F_ADD_STRINGX4_TO_BUFFER( S1:= CONCAT(sHead, '_EVP0_mA' ), S2:='$t', S3:= REAL_TO_STRING( stPropulsionCfg.aEVP_mA[0]  ), S4:='$n', wSize := wSize, pBuffer := pBuffer, wPos := wBufPos );
F_ADD_STRINGX4_TO_BUFFER( S1:= CONCAT(sHead, '_EVP1_mA' ), S2:='$t', S3:= REAL_TO_STRING( stPropulsionCfg.aEVP_mA[1]  ), S4:='$n', wSize := wSize, pBuffer := pBuffer, wPos := wBufPos );
F_ADD_STRINGX4_TO_BUFFER( S1:= CONCAT(sHead, '_EVP2_mA' ), S2:='$t', S3:= REAL_TO_STRING( stPropulsionCfg.aEVP_mA[2]  ), S4:='$n', wSize := wSize, pBuffer := pBuffer, wPos := wBufPos );
F_ADD_STRINGX4_TO_BUFFER( S1:= CONCAT(sHead, '_EVP3_mA' ), S2:='$t', S3:= REAL_TO_STRING( stPropulsionCfg.aEVP_mA[3]  ), S4:='$n', wSize := wSize, pBuffer := pBuffer, wPos := wBufPos );
F_ADD_STRINGX4_TO_BUFFER( S1:= CONCAT(sHead, '_EVP4_mA' ), S2:='$t', S3:= REAL_TO_STRING( stPropulsionCfg.aEVP_mA[4]  ), S4:='$n', wSize := wSize, pBuffer := pBuffer, wPos := wBufPos );
F_ADD_STRINGX4_TO_BUFFER( S1:= CONCAT(sHead, '_EVP5_mA' ), S2:='$t', S3:= REAL_TO_STRING( 0.0                         ), S4:='$n', wSize := wSize, pBuffer := pBuffer, wPos := wBufPos );
F_ADD_STRINGX4_TO_BUFFER( S1:= CONCAT(sHead, '_EVP6_mA' ), S2:='$t', S3:= REAL_TO_STRING( stPropulsionCfg.aEVP_mA[6]  ), S4:='$n', wSize := wSize, pBuffer := pBuffer, wPos := wBufPos );
F_ADD_STRINGX4_TO_BUFFER( S1:= CONCAT(sHead, '_EVP7_mA' ), S2:='$t', S3:= REAL_TO_STRING( stPropulsionCfg.aEVP_mA[7]  ), S4:='$n', wSize := wSize, pBuffer := pBuffer, wPos := wBufPos );
F_ADD_STRINGX4_TO_BUFFER( S1:= CONCAT(sHead, '_EVP8_mA' ), S2:='$t', S3:= REAL_TO_STRING( stPropulsionCfg.aEVP_mA[8]  ), S4:='$n', wSize := wSize, pBuffer := pBuffer, wPos := wBufPos );
F_ADD_STRINGX4_TO_BUFFER( S1:= CONCAT(sHead, '_EVP9_mA' ), S2:='$t', S3:= REAL_TO_STRING( stPropulsionCfg.aEVP_mA[9]  ), S4:='$n', wSize := wSize, pBuffer := pBuffer, wPos := wBufPos );
F_ADD_STRINGX4_TO_BUFFER( S1:= CONCAT(sHead, '_EVP10_mA'), S2:='$t', S3:= REAL_TO_STRING( stPropulsionCfg.aEVP_mA[10] ), S4:='$n', wSize := wSize, pBuffer := pBuffer, wPos := wBufPos );
END_FUNCTION

(* POU FUN/PARAMETERS/F_WRITE_SE_CYLINDER_POS_CFG, ST *)
FUNCTION F_WRITE_SE_CYLINDER_POS_CFG : BOOL
VAR_INPUT
	sHead : STRING;
	wSize   :DWORD;
	pBuffer :POINTER TO BYTE;
END_VAR
VAR_IN_OUT
	wPos     : DWORD;
	stConfig : ST_SE_CYLINDER_POS_CFG;
END_VAR
VAR
END_VAR
F_ADD_STRINGX3_TO_BUFFER( S1:= '$n#', S2:= sHead, S3:=' - Parameters:$n', wSize := wSize, pBuffer := pBuffer, wPos := wPos );

F_ADD_STRINGX4_TO_BUFFER( S1:= CONCAT(sHead, '_Ease'    ), S2:='$t', S3:= REAL_TO_STRING( stConfig.Ease    ), S4:='$n', wSize := wSize, pBuffer := pBuffer, wPos := wPos );

F_ADD_STRINGX4_TO_BUFFER( S1:= CONCAT(sHead, '_TgtLS_In'  ), S2:='$t', S3:= REAL_TO_STRING( stConfig.TgtLS_In  ), S4:='$n', wSize := wSize, pBuffer := pBuffer, wPos := wPos );
F_ADD_STRINGX4_TO_BUFFER( S1:= CONCAT(sHead, '_TgtLS_Out' ), S2:='$t', S3:= REAL_TO_STRING( stConfig.TgtLS_Out ), S4:='$n', wSize := wSize, pBuffer := pBuffer, wPos := wPos );
F_ADD_STRINGX4_TO_BUFFER( S1:= CONCAT(sHead, '_TgtLS_Slow' ), S2:='$t', S3:= REAL_TO_STRING( stConfig.TgtLS_Slow ), S4:='$n', wSize := wSize, pBuffer := pBuffer, wPos := wPos );

F_ADD_STRINGX4_TO_BUFFER( S1:= CONCAT(sHead, '_TimeMax'  ), S2:='$t', S3:= REAL_TO_STRING( stConfig.TimeMax  ), S4:='$n', wSize := wSize, pBuffer := pBuffer, wPos := wPos );
F_ADD_STRINGX4_TO_BUFFER( S1:= CONCAT(sHead, '_TimeEase' ), S2:='$t', S3:= REAL_TO_STRING( stConfig.TimeEase ), S4:='$n', wSize := wSize, pBuffer := pBuffer, wPos := wPos );

F_ADD_STRINGX4_TO_BUFFER( S1:= CONCAT(sHead, '_LS_Limit_In'  ), S2:='$t', S3:= BOOL_TO_STRING( stConfig.LS_Limit_In  ), S4:='$n', wSize := wSize, pBuffer := pBuffer, wPos := wPos );
F_ADD_STRINGX4_TO_BUFFER( S1:= CONCAT(sHead, '_LS_Limit_Out' ), S2:='$t', S3:= BOOL_TO_STRING( stConfig.LS_Limit_Out ), S4:='$n', wSize := wSize, pBuffer := pBuffer, wPos := wPos );

F_ADD_STRINGX4_TO_BUFFER( S1:= CONCAT(sHead, '_HP'  ), S2:='$t', S3:= BYTE_TO_STRING( stConfig.HP ), S4:='$n', wSize := wSize, pBuffer := pBuffer, wPos := wPos );
END_FUNCTION

(* POU FUN/PARAMETERS/F_WRITE_SE_CYLINDER_CFG, ST *)
FUNCTION F_WRITE_SE_CYLINDER_CFG : BOOL
VAR_INPUT
	sHead : STRING;
	wSize   :DWORD;
	pBuffer :POINTER TO BYTE;
END_VAR
VAR_IN_OUT
	wPos     : DWORD;
	stConfig : ST_SE_CYLINDER_CFG;
END_VAR
VAR
END_VAR
F_ADD_STRINGX3_TO_BUFFER( S1:= '$n#', S2:= sHead, S3:=' - Parameters:$n', wSize := wSize, pBuffer := pBuffer, wPos := wPos );

F_ADD_STRINGX4_TO_BUFFER( S1:= CONCAT(sHead, '_Ease'     ), S2:='$t', S3:= REAL_TO_STRING( stConfig.Ease     ), S4:='$n', wSize := wSize, pBuffer := pBuffer, wPos := wPos );
F_ADD_STRINGX4_TO_BUFFER( S1:= CONCAT(sHead, '_TimeMax'  ), S2:='$t', S3:= REAL_TO_STRING( stConfig.TimeMax  ), S4:='$n', wSize := wSize, pBuffer := pBuffer, wPos := wPos );
F_ADD_STRINGX4_TO_BUFFER( S1:= CONCAT(sHead, '_TimeEase' ), S2:='$t', S3:= REAL_TO_STRING( stConfig.TimeEase ), S4:='$n', wSize := wSize, pBuffer := pBuffer, wPos := wPos );
F_ADD_STRINGX4_TO_BUFFER( S1:= CONCAT(sHead, '_HP'       ), S2:='$t', S3:= BYTE_TO_STRING( stConfig.HP       ), S4:='$n', wSize := wSize, pBuffer := pBuffer, wPos := wPos );
END_FUNCTION

(* POU FUN/PARAMETERS/F_WRITE_LIFT_PROP_CFG, ST *)
FUNCTION F_WRITE_LIFT_PROP_CFG : BOOL
VAR_INPUT
	sHead : STRING;
	wSize   :DWORD;
	pBuffer :POINTER TO BYTE;
END_VAR
VAR_IN_OUT
	wPos     : DWORD;
	stConfig : ST_LIFT_PROP_CFG;
END_VAR
VAR
END_VAR
F_ADD_STRINGX3_TO_BUFFER( S1:= '$n#', S2:= sHead, S3:=' - Parameters:$n', wSize := wSize, pBuffer := pBuffer, wPos := wPos );

F_ADD_STRINGX4_TO_BUFFER( S1:= CONCAT(sHead, '_TgtP_Up'  ), S2:='$t', S3:= REAL_TO_STRING( stConfig.TgtP_Up  ), S4:='$n', wSize := wSize, pBuffer := pBuffer, wPos := wPos );
F_ADD_STRINGX4_TO_BUFFER( S1:= CONCAT(sHead, '_TgtP_Dw'  ), S2:='$t', S3:= REAL_TO_STRING( stConfig.TgtP_Dw  ), S4:='$n', wSize := wSize, pBuffer := pBuffer, wPos := wPos );
F_ADD_STRINGX4_TO_BUFFER( S1:= CONCAT(sHead, '_TgtLS_Up' ), S2:='$t', S3:= REAL_TO_STRING( stConfig.TgtLS_Up ), S4:='$n', wSize := wSize, pBuffer := pBuffer, wPos := wPos );
F_ADD_STRINGX4_TO_BUFFER( S1:= CONCAT(sHead, '_TgtLS_Dw' ), S2:='$t', S3:= REAL_TO_STRING( stConfig.TgtLS_Dw ), S4:='$n', wSize := wSize, pBuffer := pBuffer, wPos := wPos );

F_ADD_STRINGX4_TO_BUFFER( S1:= CONCAT(sHead, '_P_DB'     ), S2:='$t', S3:= REAL_TO_STRING( stConfig.P_DB     ), S4:='$n', wSize := wSize, pBuffer := pBuffer, wPos := wPos );
F_ADD_STRINGX4_TO_BUFFER( S1:= CONCAT(sHead, '_LS_DB'    ), S2:='$t', S3:= REAL_TO_STRING( stConfig.LS_DB    ), S4:='$n', wSize := wSize, pBuffer := pBuffer, wPos := wPos );

F_ADD_STRINGX4_TO_BUFFER( S1:= CONCAT(sHead, '_TimeMax'  ), S2:='$t', S3:= REAL_TO_STRING( stConfig.TimeMax  ), S4:='$n', wSize := wSize, pBuffer := pBuffer, wPos := wPos );
F_ADD_STRINGX4_TO_BUFFER( S1:= CONCAT(sHead, '_Delay_Up' ), S2:='$t', S3:= REAL_TO_STRING( stConfig.Delay_Up ), S4:='$n', wSize := wSize, pBuffer := pBuffer, wPos := wPos );
F_ADD_STRINGX4_TO_BUFFER( S1:= CONCAT(sHead, '_Delay_Dw' ), S2:='$t', S3:= REAL_TO_STRING( stConfig.Delay_Dw ), S4:='$n', wSize := wSize, pBuffer := pBuffer, wPos := wPos );

F_ADD_STRINGX4_TO_BUFFER( S1:= CONCAT(sHead, '_HP_Up'  ), S2:='$t', S3:= BYTE_TO_STRING( stConfig.HP_Up ), S4:='$n', wSize := wSize, pBuffer := pBuffer, wPos := wPos );
F_ADD_STRINGX4_TO_BUFFER( S1:= CONCAT(sHead, '_HP_Dw'  ), S2:='$t', S3:= BYTE_TO_STRING( stConfig.HP_Dw ), S4:='$n', wSize := wSize, pBuffer := pBuffer, wPos := wPos );
END_FUNCTION

(* POU FUN/PARAMETERS/F_WRITE_DE_CYLINDER_POS_CFG, ST *)
FUNCTION F_WRITE_DE_CYLINDER_POS_CFG : BOOL
VAR_INPUT
	sHead : STRING;
	wSize   :DWORD;
	pBuffer :POINTER TO BYTE;
END_VAR
VAR_IN_OUT
	wPos     : DWORD;
	stConfig : ST_DE_CYLINDER_POS_CFG;
END_VAR
VAR
END_VAR
F_ADD_STRINGX3_TO_BUFFER( S1:= '$n#', S2:= sHead, S3:=' - Parameters:$n', wSize := wSize, pBuffer := pBuffer, wPos := wPos );

F_ADD_STRINGX4_TO_BUFFER( S1:= CONCAT(sHead, '_TgtLS_In'  ), S2:='$t', S3:= REAL_TO_STRING( stConfig.TgtLS_In  ), S4:='$n', wSize := wSize, pBuffer := pBuffer, wPos := wPos );
F_ADD_STRINGX4_TO_BUFFER( S1:= CONCAT(sHead, '_TgtLS_Out' ), S2:='$t', S3:= REAL_TO_STRING( stConfig.TgtLS_Out ), S4:='$n', wSize := wSize, pBuffer := pBuffer, wPos := wPos );
F_ADD_STRINGX4_TO_BUFFER( S1:= CONCAT(sHead, '_TgtLS_Mid' ), S2:='$t', S3:= REAL_TO_STRING( stConfig.TgtLS_Mid ), S4:='$n', wSize := wSize, pBuffer := pBuffer, wPos := wPos );
F_ADD_STRINGX4_TO_BUFFER( S1:= CONCAT(sHead, '_TgtLS_DB'  ), S2:='$t', S3:= REAL_TO_STRING( stConfig.TgtLS_DB  ), S4:='$n', wSize := wSize, pBuffer := pBuffer, wPos := wPos );

F_ADD_STRINGX4_TO_BUFFER( S1:= CONCAT(sHead, '_TimeMax'  ), S2:='$t', S3:= REAL_TO_STRING( stConfig.TimeMax  ), S4:='$n', wSize := wSize, pBuffer := pBuffer, wPos := wPos );

F_ADD_STRINGX4_TO_BUFFER( S1:= CONCAT(sHead, '_LS_Limit_In'  ), S2:='$t', S3:= BOOL_TO_STRING( stConfig.LS_Limit_In  ), S4:='$n', wSize := wSize, pBuffer := pBuffer, wPos := wPos );
F_ADD_STRINGX4_TO_BUFFER( S1:= CONCAT(sHead, '_LS_Limit_Out' ), S2:='$t', S3:= BOOL_TO_STRING( stConfig.LS_Limit_Out ), S4:='$n', wSize := wSize, pBuffer := pBuffer, wPos := wPos );

F_ADD_STRINGX4_TO_BUFFER( S1:= CONCAT(sHead, '_HP'  ), S2:='$t', S3:= BYTE_TO_STRING( stConfig.HP ), S4:='$n', wSize := wSize, pBuffer := pBuffer, wPos := wPos );
END_FUNCTION

(* POU FUN/PARAMETERS/F_WRITE_WB_CFG, ST *)
FUNCTION F_WRITE_WB_CFG : BOOL
VAR_INPUT
	sHead : STRING;
	wSize   :DWORD;
	pBuffer :POINTER TO BYTE;
END_VAR
VAR_IN_OUT
	wPos     : DWORD;
	stConfig : ST_WB_CFG;
END_VAR
VAR
END_VAR
F_ADD_STRINGX3_TO_BUFFER( S1:= '$n#', S2:= sHead, S3:=' - Parameters:$n', wSize := wSize, pBuffer := pBuffer, wPos := wPos );

F_ADD_STRINGX4_TO_BUFFER( S1:= CONCAT(sHead, '_TimeMax_Idle'   ), S2:='$t', S3:= REAL_TO_STRING( stConfig.TimeMax_Idle  ), S4:='$n', wSize := wSize, pBuffer := pBuffer, wPos := wPos );
F_ADD_STRINGX4_TO_BUFFER( S1:= CONCAT(sHead, '_TimeMax_Init'   ), S2:='$t', S3:= REAL_TO_STRING( stConfig.TimeMax_Init  ), S4:='$n', wSize := wSize, pBuffer := pBuffer, wPos := wPos );
F_ADD_STRINGX4_TO_BUFFER( S1:= CONCAT(sHead, '_TimeMax_DumpFwd'   ), S2:='$t', S3:= REAL_TO_STRING( stConfig.TimeMax_DumpFwd  ), S4:='$n', wSize := wSize, pBuffer := pBuffer, wPos := wPos );
F_ADD_STRINGX4_TO_BUFFER( S1:= CONCAT(sHead, '_TimeMax_DumpAft'   ), S2:='$t', S3:= REAL_TO_STRING( stConfig.TimeMax_DumpAft  ), S4:='$n', wSize := wSize, pBuffer := pBuffer, wPos := wPos );
F_ADD_STRINGX4_TO_BUFFER( S1:= CONCAT(sHead, '_TimeMax_MoveFwd'   ), S2:='$t', S3:= REAL_TO_STRING( stConfig.TimeMax_MoveFwd  ), S4:='$n', wSize := wSize, pBuffer := pBuffer, wPos := wPos );
F_ADD_STRINGX4_TO_BUFFER( S1:= CONCAT(sHead, '_TimeMax_MoveAft'   ), S2:='$t', S3:= REAL_TO_STRING( stConfig.TimeMax_MoveAft  ), S4:='$n', wSize := wSize, pBuffer := pBuffer, wPos := wPos );

F_ADD_STRINGX4_TO_BUFFER( S1:= CONCAT(sHead, '_EVP_Pump_Min' ), S2:='$t', S3:= REAL_TO_STRING( stConfig.EVP_Pump_Min ), S4:='$n', wSize := wSize, pBuffer := pBuffer, wPos := wPos );
F_ADD_STRINGX4_TO_BUFFER( S1:= CONCAT(sHead, '_EVP_Pump_Max' ), S2:='$t', S3:= REAL_TO_STRING( stConfig.EVP_Pump_Max ), S4:='$n', wSize := wSize, pBuffer := pBuffer, wPos := wPos );
F_ADD_STRINGX4_TO_BUFFER( S1:= CONCAT(sHead, '_EVP_Pump_Inc' ), S2:='$t', S3:= REAL_TO_STRING( stConfig.EVP_Pump_Inc ), S4:='$n', wSize := wSize, pBuffer := pBuffer, wPos := wPos );
F_ADD_STRINGX4_TO_BUFFER( S1:= CONCAT(sHead, '_EVP_Pump_Dec' ), S2:='$t', S3:= REAL_TO_STRING( stConfig.EVP_Pump_Dec ), S4:='$n', wSize := wSize, pBuffer := pBuffer, wPos := wPos );

F_ADD_STRINGX4_TO_BUFFER( S1:= CONCAT(sHead, '_LP'        ), S2:='$t', S3:= BYTE_TO_STRING( stConfig.LP        ), S4:='$n', wSize := wSize, pBuffer := pBuffer, wPos := wPos );

F_ADD_STRINGX4_TO_BUFFER( S1:= CONCAT(sHead, '_EnScoopAF' ), S2:='$t', S3:= BOOL_TO_STRING( stConfig.EnScoopAF ), S4:='$n', wSize := wSize, pBuffer := pBuffer, wPos := wPos );
END_FUNCTION

(* POU FUN/PARAMETERS/F_WRITE_WB_VALVESF_CFG, ST *)
FUNCTION F_WRITE_WB_VALVESF_CFG : BOOL
VAR_INPUT
	sHead : STRING;
	wSize   :DWORD;
	pBuffer :POINTER TO BYTE;
END_VAR
VAR_IN_OUT
	wPos     : DWORD;
	stConfig : ST_WB_VALVE_CFG;
END_VAR
VAR
END_VAR
F_ADD_STRINGX3_TO_BUFFER( S1:= '$n#', S2:= sHead, S3:=' - Parameters:$n', wSize := wSize, pBuffer := pBuffer, wPos := wPos );

F_ADD_STRINGX4_TO_BUFFER( S1:= CONCAT(sHead, '_TimeMax'   ), S2:='$t', S3:= REAL_TO_STRING( stConfig.TimeMax  ), S4:='$n', wSize := wSize, pBuffer := pBuffer, wPos := wPos );
F_ADD_STRINGX4_TO_BUFFER( S1:= CONCAT(sHead, '_PushTime'  ), S2:='$t', S3:= REAL_TO_STRING( stConfig.PushTime ), S4:='$n', wSize := wSize, pBuffer := pBuffer, wPos := wPos );
F_ADD_STRINGX4_TO_BUFFER( S1:= CONCAT(sHead, '_PushPress' ), S2:='$t', S3:= REAL_TO_STRING( stConfig.PushP    ), S4:='$n', wSize := wSize, pBuffer := pBuffer, wPos := wPos );
F_ADD_STRINGX4_TO_BUFFER( S1:= CONCAT(sHead, '_HP'        ), S2:='$t', S3:= BYTE_TO_STRING( stConfig.HP       ), S4:='$n', wSize := wSize, pBuffer := pBuffer, wPos := wPos );
END_FUNCTION

(* POU FUN/PARAMETERS/F_WRITE_WB_VALVELS_CFG, ST *)
FUNCTION F_WRITE_WB_VALVELS_CFG : BOOL
VAR_INPUT
	sHead : STRING;
	wSize   :DWORD;
	pBuffer :POINTER TO BYTE;
END_VAR
VAR_IN_OUT
	wPos     : DWORD;
	stConfig : ST_WB_VALVE_LS_CFG;
END_VAR
VAR
END_VAR
F_ADD_STRINGX3_TO_BUFFER( S1:= '$n#', S2:= sHead, S3:=' - Parameters:$n', wSize := wSize, pBuffer := pBuffer, wPos := wPos );

F_ADD_STRINGX4_TO_BUFFER( S1:= CONCAT(sHead, '_TimeMax'   ), S2:='$t', S3:= REAL_TO_STRING( stConfig.TimeMax  ), S4:='$n', wSize := wSize, pBuffer := pBuffer, wPos := wPos );
F_ADD_STRINGX4_TO_BUFFER( S1:= CONCAT(sHead, '_PushTime'  ), S2:='$t', S3:= REAL_TO_STRING( stConfig.PushTime ), S4:='$n', wSize := wSize, pBuffer := pBuffer, wPos := wPos );
F_ADD_STRINGX4_TO_BUFFER( S1:= CONCAT(sHead, '_PushPress' ), S2:='$t', S3:= REAL_TO_STRING( stConfig.PushP    ), S4:='$n', wSize := wSize, pBuffer := pBuffer, wPos := wPos );

F_ADD_STRINGX4_TO_BUFFER( S1:= CONCAT(sHead, '_TgtLS_Half' ), S2:='$t', S3:= REAL_TO_STRING( stConfig.TgtLS_Half ), S4:='$n', wSize := wSize, pBuffer := pBuffer, wPos := wPos );
F_ADD_STRINGX4_TO_BUFFER( S1:= CONCAT(sHead, '_LS_DB'      ), S2:='$t', S3:= REAL_TO_STRING( stConfig.LS_DB      ), S4:='$n', wSize := wSize, pBuffer := pBuffer, wPos := wPos );

F_ADD_STRINGX4_TO_BUFFER( S1:= CONCAT(sHead, '_HP'        ), S2:='$t', S3:= BYTE_TO_STRING( stConfig.HP       ), S4:='$n', wSize := wSize, pBuffer := pBuffer, wPos := wPos );
END_FUNCTION

(* POU FUN/PARAMETERS/F_WRITE_WINCHE_CFG, ST *)
FUNCTION F_WRITE_WINCHE_CFG : BOOL
VAR_INPUT
	sHead : STRING;
	wSize   :DWORD;
	pBuffer :POINTER TO BYTE;
END_VAR
VAR_IN_OUT
	wPos     : DWORD;
	stConfig : ST_WINCHE_CFG;
END_VAR
VAR
	aux1 : REAL;
	aux2 : REAL;
	aux3 : REAL;
END_VAR
F_ADD_STRINGX3_TO_BUFFER( S1:= '$n#', S2:= sHead, S3:=' - Parameters:$n', wSize := wSize, pBuffer := pBuffer, wPos := wPos );

F_ADD_STRINGX4_TO_BUFFER( S1:= CONCAT(sHead, '_Spd11' ), S2:='$t', S3:= REAL_TO_STRING( stConfig.Spd1[1] ), S4:='$n', wSize := wSize, pBuffer := pBuffer, wPos := wPos );
F_ADD_STRINGX4_TO_BUFFER( S1:= CONCAT(sHead, '_Spd21' ), S2:='$t', S3:= REAL_TO_STRING( stConfig.Spd2[1] ), S4:='$n', wSize := wSize, pBuffer := pBuffer, wPos := wPos );
F_ADD_STRINGX4_TO_BUFFER( S1:= CONCAT(sHead, '_Spd31' ), S2:='$t', S3:= REAL_TO_STRING( stConfig.Spd3[1] ), S4:='$n', wSize := wSize, pBuffer := pBuffer, wPos := wPos );

F_ADD_STRINGX4_TO_BUFFER( S1:= CONCAT(sHead, '_Spd17' ), S2:='$t', S3:= REAL_TO_STRING( stConfig.Spd1[7] ), S4:='$n', wSize := wSize, pBuffer := pBuffer, wPos := wPos );
F_ADD_STRINGX4_TO_BUFFER( S1:= CONCAT(sHead, '_Spd27' ), S2:='$t', S3:= REAL_TO_STRING( stConfig.Spd2[7] ), S4:='$n', wSize := wSize, pBuffer := pBuffer, wPos := wPos );
F_ADD_STRINGX4_TO_BUFFER( S1:= CONCAT(sHead, '_Spd37' ), S2:='$t', S3:= REAL_TO_STRING( stConfig.Spd3[7] ), S4:='$n', wSize := wSize, pBuffer := pBuffer, wPos := wPos );

F_ADD_STRINGX4_TO_BUFFER( S1:= CONCAT(sHead, '_P1_Max' ), S2:='$t', S3:= REAL_TO_STRING( stConfig.P1_Max ), S4:='$n', wSize := wSize, pBuffer := pBuffer, wPos := wPos );
F_ADD_STRINGX4_TO_BUFFER( S1:= CONCAT(sHead, '_P2_Max' ), S2:='$t', S3:= REAL_TO_STRING( stConfig.P2_Max ), S4:='$n', wSize := wSize, pBuffer := pBuffer, wPos := wPos );
F_ADD_STRINGX4_TO_BUFFER( S1:= CONCAT(sHead, '_P3_Max' ), S2:='$t', S3:= REAL_TO_STRING( stConfig.P3_Max ), S4:='$n', wSize := wSize, pBuffer := pBuffer, wPos := wPos );

F_ADD_STRINGX4_TO_BUFFER( S1:= CONCAT(sHead, '_A_Spd1' ), S2:='$t', S3:= BOOL_TO_STRING( stConfig.A_Spd1 ), S4:='$n', wSize := wSize, pBuffer := pBuffer, wPos := wPos );

F_ADD_STRINGX4_TO_BUFFER( S1:= CONCAT(sHead, '_TimeMax' ), S2:='$t', S3:= REAL_TO_STRING( stConfig.TimeMax ), S4:='$n', wSize := wSize, pBuffer := pBuffer, wPos := wPos );

(*F_ADD_STRINGX4_TO_BUFFER( S1:= CONCAT(sHead, '_PP'  ), S2:='$t', S3:= BYTE_TO_STRING( stConfig.PP ), S4:='$n', wSize := wSize, pBuffer := pBuffer, wPos := wPos );*)

(*Calc Values*)

aux1 := (stConfig.Spd1[7]-stConfig.Spd1[1])/6.0;
aux2 := (stConfig.Spd2[7]-stConfig.Spd2[1])/6.0;
aux3 := (stConfig.Spd3[7]-stConfig.Spd3[1])/6.0;

stConfig.Spd1[2] := stConfig.Spd1[1] + Aux1;
stConfig.Spd1[3] := stConfig.Spd1[2] + Aux1;
stConfig.Spd1[4] := stConfig.Spd1[3] + Aux1;
stConfig.Spd1[5] := stConfig.Spd1[4] + Aux1;
stConfig.Spd1[6] := stConfig.Spd1[5] + Aux1;

stConfig.Spd2[2] := stConfig.Spd2[1] + Aux2;
stConfig.Spd2[3] := stConfig.Spd2[2] + Aux2;
stConfig.Spd2[4] := stConfig.Spd2[3] + Aux2;
stConfig.Spd2[5] := stConfig.Spd2[4] + Aux2;
stConfig.Spd2[6] := stConfig.Spd2[5] + Aux2;

stConfig.Spd3[2] := stConfig.Spd3[1] + Aux3;
stConfig.Spd3[3] := stConfig.Spd3[2] + Aux3;
stConfig.Spd3[4] := stConfig.Spd3[3] + Aux3;
stConfig.Spd3[5] := stConfig.Spd3[4] + Aux3;
stConfig.Spd3[6] := stConfig.Spd3[5] + Aux3;
END_FUNCTION

(* POU FUN/PARAMETERS/F_WRITE_BOARD_CFG, ST *)
FUNCTION F_WRITE_BOARD_CFG : BOOL
VAR_INPUT
	sHead : STRING;
	wSize   :DWORD;
	pBuffer :POINTER TO BYTE;
END_VAR
VAR_IN_OUT
	wPos     : DWORD;
	stConfig : ST_BOARD_CFG;
END_VAR
VAR
END_VAR
F_ADD_STRINGX3_TO_BUFFER( S1:= '$n#', S2:= sHead, S3:=' - Parameters:$n', wSize := wSize, pBuffer := pBuffer, wPos := wPos );

F_ADD_STRINGX4_TO_BUFFER( S1:= CONCAT(sHead, '_TgtLS_P_In'   ), S2:='$t', S3:= REAL_TO_STRING( stConfig.TgtLS_P_In   ), S4:='$n', wSize := wSize, pBuffer := pBuffer, wPos := wPos );
F_ADD_STRINGX4_TO_BUFFER( S1:= CONCAT(sHead, '_TgtLS_P_InR'  ), S2:='$t', S3:= REAL_TO_STRING( stConfig.TgtLS_P_InR  ), S4:='$n', wSize := wSize, pBuffer := pBuffer, wPos := wPos );
F_ADD_STRINGX4_TO_BUFFER( S1:= CONCAT(sHead, '_TgtLS_P_Out'  ), S2:='$t', S3:= REAL_TO_STRING( stConfig.TgtLS_P_Out  ), S4:='$n', wSize := wSize, pBuffer := pBuffer, wPos := wPos );
F_ADD_STRINGX4_TO_BUFFER( S1:= CONCAT(sHead, '_TgtLS_P_OutR' ), S2:='$t', S3:= REAL_TO_STRING( stConfig.TgtLS_P_OutR ), S4:='$n', wSize := wSize, pBuffer := pBuffer, wPos := wPos );
F_ADD_STRINGX4_TO_BUFFER( S1:= CONCAT(sHead, '_TgtLS_P_Mid'  ), S2:='$t', S3:= REAL_TO_STRING( stConfig.TgtLS_P_Mid  ), S4:='$n', wSize := wSize, pBuffer := pBuffer, wPos := wPos );

F_ADD_STRINGX4_TO_BUFFER( S1:= CONCAT(sHead, '_TgtLS_S_In'   ), S2:='$t', S3:= REAL_TO_STRING( stConfig.TgtLS_S_In   ), S4:='$n', wSize := wSize, pBuffer := pBuffer, wPos := wPos );
F_ADD_STRINGX4_TO_BUFFER( S1:= CONCAT(sHead, '_TgtLS_S_InR'  ), S2:='$t', S3:= REAL_TO_STRING( stConfig.TgtLS_S_InR  ), S4:='$n', wSize := wSize, pBuffer := pBuffer, wPos := wPos );
F_ADD_STRINGX4_TO_BUFFER( S1:= CONCAT(sHead, '_TgtLS_S_Out'  ), S2:='$t', S3:= REAL_TO_STRING( stConfig.TgtLS_S_Out  ), S4:='$n', wSize := wSize, pBuffer := pBuffer, wPos := wPos );
F_ADD_STRINGX4_TO_BUFFER( S1:= CONCAT(sHead, '_TgtLS_S_OutR' ), S2:='$t', S3:= REAL_TO_STRING( stConfig.TgtLS_S_OutR ), S4:='$n', wSize := wSize, pBuffer := pBuffer, wPos := wPos );
F_ADD_STRINGX4_TO_BUFFER( S1:= CONCAT(sHead, '_TgtLS_S_Mid'  ), S2:='$t', S3:= REAL_TO_STRING( stConfig.TgtLS_S_Mid  ), S4:='$n', wSize := wSize, pBuffer := pBuffer, wPos := wPos );

F_ADD_STRINGX4_TO_BUFFER( S1:= CONCAT(sHead, '_TgtLS_P_Safe_In'  ), S2:='$t', S3:= REAL_TO_STRING( stConfig.TgtLS_P_Safe_In  ), S4:='$n', wSize := wSize, pBuffer := pBuffer, wPos := wPos );
F_ADD_STRINGX4_TO_BUFFER( S1:= CONCAT(sHead, '_TgtLS_P_Safe_Out' ), S2:='$t', S3:= REAL_TO_STRING( stConfig.TgtLS_P_Safe_Out ), S4:='$n', wSize := wSize, pBuffer := pBuffer, wPos := wPos );

F_ADD_STRINGX4_TO_BUFFER( S1:= CONCAT(sHead, '_TgtLS_S_Safe_In'  ), S2:='$t', S3:= REAL_TO_STRING( stConfig.TgtLS_S_Safe_In  ), S4:='$n', wSize := wSize, pBuffer := pBuffer, wPos := wPos );
F_ADD_STRINGX4_TO_BUFFER( S1:= CONCAT(sHead, '_TgtLS_S_Safe_Out' ), S2:='$t', S3:= REAL_TO_STRING( stConfig.TgtLS_S_Safe_Out ), S4:='$n', wSize := wSize, pBuffer := pBuffer, wPos := wPos );

F_ADD_STRINGX4_TO_BUFFER( S1:= CONCAT(sHead, '_LS_Dif_Tgt' ), S2:='$t', S3:= REAL_TO_STRING( stConfig.LS_Dif_Tgt ), S4:='$n', wSize := wSize, pBuffer := pBuffer, wPos := wPos );
F_ADD_STRINGX4_TO_BUFFER( S1:= CONCAT(sHead, '_LS_Dif_Max' ), S2:='$t', S3:= REAL_TO_STRING( stConfig.LS_Dif_Max ), S4:='$n', wSize := wSize, pBuffer := pBuffer, wPos := wPos );
F_ADD_STRINGX4_TO_BUFFER( S1:= CONCAT(sHead, '_LS_Dif_Min' ), S2:='$t', S3:= REAL_TO_STRING( stConfig.LS_Dif_Min ), S4:='$n', wSize := wSize, pBuffer := pBuffer, wPos := wPos );

F_ADD_STRINGX4_TO_BUFFER( S1:= CONCAT(sHead, '_LS_DB'   ), S2:='$t', S3:= REAL_TO_STRING( stConfig.LS_DB   ), S4:='$n', wSize := wSize, pBuffer := pBuffer, wPos := wPos );

F_ADD_STRINGX4_TO_BUFFER( S1:= CONCAT(sHead, '_P_Hyst_HP' ), S2:='$t', S3:= REAL_TO_STRING( stConfig.P_Hyst_HP ), S4:='$n', wSize := wSize, pBuffer := pBuffer, wPos := wPos );
F_ADD_STRINGX4_TO_BUFFER( S1:= CONCAT(sHead, '_P_Hyst_LP' ), S2:='$t', S3:= REAL_TO_STRING( stConfig.P_Hyst_LP ), S4:='$n', wSize := wSize, pBuffer := pBuffer, wPos := wPos );
F_ADD_STRINGX4_TO_BUFFER( S1:= CONCAT(sHead, '_P_Hyst_TM' ), S2:='$t', S3:= REAL_TO_STRING( stConfig.P_Hyst_TM ), S4:='$n', wSize := wSize, pBuffer := pBuffer, wPos := wPos );

(*Keel Limits*)
F_ADD_STRINGX4_TO_BUFFER( S1:= CONCAT(sHead, '_Keel_P_Max' ), S2:='$t', S3:= REAL_TO_STRING( stConfig.Keel_P_Max ), S4:='$n', wSize := wSize, pBuffer := pBuffer, wPos := wPos );
F_ADD_STRINGX4_TO_BUFFER( S1:= CONCAT(sHead, '_Keel_S_Min' ), S2:='$t', S3:= REAL_TO_STRING( stConfig.Keel_S_Min ), S4:='$n', wSize := wSize, pBuffer := pBuffer, wPos := wPos );

(*Valve Limits*)
F_ADD_STRINGX4_TO_BUFFER( S1:= CONCAT(sHead, '_EVP_In_P_Min' ), S2:='$t', S3:= REAL_TO_STRING( stConfig.EVP_In_P_Min ), S4:='$n', wSize := wSize, pBuffer := pBuffer, wPos := wPos );
F_ADD_STRINGX4_TO_BUFFER( S1:= CONCAT(sHead, '_EVP_In_P_Max' ), S2:='$t', S3:= REAL_TO_STRING( stConfig.EVP_In_P_Max ), S4:='$n', wSize := wSize, pBuffer := pBuffer, wPos := wPos );

F_ADD_STRINGX4_TO_BUFFER( S1:= CONCAT(sHead, '_EVP_In_S_Min' ), S2:='$t', S3:= REAL_TO_STRING( stConfig.EVP_In_S_Min ), S4:='$n', wSize := wSize, pBuffer := pBuffer, wPos := wPos );
F_ADD_STRINGX4_TO_BUFFER( S1:= CONCAT(sHead, '_EVP_In_S_Max' ), S2:='$t', S3:= REAL_TO_STRING( stConfig.EVP_In_S_Max ), S4:='$n', wSize := wSize, pBuffer := pBuffer, wPos := wPos );

F_ADD_STRINGX4_TO_BUFFER( S1:= CONCAT(sHead, '_EVP_Out_P_Min' ), S2:='$t', S3:= REAL_TO_STRING( stConfig.EVP_Out_P_Min ), S4:='$n', wSize := wSize, pBuffer := pBuffer, wPos := wPos );
F_ADD_STRINGX4_TO_BUFFER( S1:= CONCAT(sHead, '_EVP_Out_P_Max' ), S2:='$t', S3:= REAL_TO_STRING( stConfig.EVP_Out_P_Max ), S4:='$n', wSize := wSize, pBuffer := pBuffer, wPos := wPos );

F_ADD_STRINGX4_TO_BUFFER( S1:= CONCAT(sHead, '_EVP_Out_S_Min' ), S2:='$t', S3:= REAL_TO_STRING( stConfig.EVP_Out_S_Min ), S4:='$n', wSize := wSize, pBuffer := pBuffer, wPos := wPos );
F_ADD_STRINGX4_TO_BUFFER( S1:= CONCAT(sHead, '_EVP_Out_S_Max' ), S2:='$t', S3:= REAL_TO_STRING( stConfig.EVP_Out_S_Max ), S4:='$n', wSize := wSize, pBuffer := pBuffer, wPos := wPos );

(*Valve Targets*)
F_ADD_STRINGX4_TO_BUFFER( S1:= CONCAT(sHead, '_EVP_In_P_Eng' ), S2:='$t', S3:= REAL_TO_STRING( stConfig.EVP_In_P_Eng ), S4:='$n', wSize := wSize, pBuffer := pBuffer, wPos := wPos );
F_ADD_STRINGX4_TO_BUFFER( S1:= CONCAT(sHead, '_EVP_In_P_PP'  ), S2:='$t', S3:= REAL_TO_STRING( stConfig.EVP_In_P_PP  ), S4:='$n', wSize := wSize, pBuffer := pBuffer, wPos := wPos );

F_ADD_STRINGX4_TO_BUFFER( S1:= CONCAT(sHead, '_EVP_In_S_Eng' ), S2:='$t', S3:= REAL_TO_STRING( stConfig.EVP_In_S_Eng ), S4:='$n', wSize := wSize, pBuffer := pBuffer, wPos := wPos );
F_ADD_STRINGX4_TO_BUFFER( S1:= CONCAT(sHead, '_EVP_In_S_PP'  ), S2:='$t', S3:= REAL_TO_STRING( stConfig.EVP_In_S_PP  ), S4:='$n', wSize := wSize, pBuffer := pBuffer, wPos := wPos );

F_ADD_STRINGX4_TO_BUFFER( S1:= CONCAT(sHead, '_EVP_Out_P_Eng' ), S2:='$t', S3:= REAL_TO_STRING( stConfig.EVP_Out_P_Eng ), S4:='$n', wSize := wSize, pBuffer := pBuffer, wPos := wPos );
F_ADD_STRINGX4_TO_BUFFER( S1:= CONCAT(sHead, '_EVP_Out_P_PP'  ), S2:='$t', S3:= REAL_TO_STRING( stConfig.EVP_Out_P_PP  ), S4:='$n', wSize := wSize, pBuffer := pBuffer, wPos := wPos );

F_ADD_STRINGX4_TO_BUFFER( S1:= CONCAT(sHead, '_EVP_Out_S_Eng' ), S2:='$t', S3:= REAL_TO_STRING( stConfig.EVP_Out_S_Eng ), S4:='$n', wSize := wSize, pBuffer := pBuffer, wPos := wPos );
F_ADD_STRINGX4_TO_BUFFER( S1:= CONCAT(sHead, '_EVP_Out_S_PP'  ), S2:='$t', S3:= REAL_TO_STRING( stConfig.EVP_Out_S_PP  ), S4:='$n', wSize := wSize, pBuffer := pBuffer, wPos := wPos );


(*Valve Gains*)
F_ADD_STRINGX4_TO_BUFFER( S1:= CONCAT(sHead, '_EVP_In_EVP_K'  ), S2:='$t', S3:= REAL_TO_STRING( stConfig.EVP_In_EVP_K  ), S4:='$n', wSize := wSize, pBuffer := pBuffer, wPos := wPos );
F_ADD_STRINGX4_TO_BUFFER( S1:= CONCAT(sHead, '_EVP_Out_EVP_K' ), S2:='$t', S3:= REAL_TO_STRING( stConfig.EVP_Out_EVP_K ), S4:='$n', wSize := wSize, pBuffer := pBuffer, wPos := wPos );

F_ADD_STRINGX4_TO_BUFFER( S1:= CONCAT(sHead, '_EVP_In_LS_K'  ), S2:='$t', S3:= REAL_TO_STRING( stConfig.EVP_In_LS_K  ), S4:='$n', wSize := wSize, pBuffer := pBuffer, wPos := wPos );
F_ADD_STRINGX4_TO_BUFFER( S1:= CONCAT(sHead, '_EVP_Out_LS_K' ), S2:='$t', S3:= REAL_TO_STRING( stConfig.EVP_Out_LS_K ), S4:='$n', wSize := wSize, pBuffer := pBuffer, wPos := wPos );

(*Valve Softstart*)
F_ADD_STRINGX4_TO_BUFFER( S1:= CONCAT(sHead, '_EVP_In_Inc'  ), S2:='$t', S3:= REAL_TO_STRING( stConfig.EVP_In_Inc  ), S4:='$n', wSize := wSize, pBuffer := pBuffer, wPos := wPos );
F_ADD_STRINGX4_TO_BUFFER( S1:= CONCAT(sHead, '_EVP_Out_Inc' ), S2:='$t', S3:= REAL_TO_STRING( stConfig.EVP_Out_Inc ), S4:='$n', wSize := wSize, pBuffer := pBuffer, wPos := wPos );

F_ADD_STRINGX4_TO_BUFFER( S1:= CONCAT(sHead, '_EVP_In_Dec'  ), S2:='$t', S3:= REAL_TO_STRING( stConfig.EVP_In_Dec  ), S4:='$n', wSize := wSize, pBuffer := pBuffer, wPos := wPos );
F_ADD_STRINGX4_TO_BUFFER( S1:= CONCAT(sHead, '_EVP_Out_Dec' ), S2:='$t', S3:= REAL_TO_STRING( stConfig.EVP_Out_Dec ), S4:='$n', wSize := wSize, pBuffer := pBuffer, wPos := wPos );

F_ADD_STRINGX4_TO_BUFFER( S1:= CONCAT(sHead, '_LP'  ), S2:='$t', S3:= BYTE_TO_STRING( stConfig.LP ), S4:='$n', wSize := wSize, pBuffer := pBuffer, wPos := wPos );

F_ADD_STRINGX4_TO_BUFFER( S1:= CONCAT(sHead, '_TimeMax'  ), S2:='$t', S3:= REAL_TO_STRING( stConfig.TimeMax  ), S4:='$n', wSize := wSize, pBuffer := pBuffer, wPos := wPos );
END_FUNCTION

(* POU FUN/PARAMETERS/F_WRITE_KEEL_CFG, ST *)
FUNCTION F_WRITE_KEEL_CFG : BOOL
VAR_INPUT
	sHead   : STRING;
	wSize   :DWORD;
	pBuffer :POINTER TO BYTE;
END_VAR
VAR_IN_OUT
	wPos     : DWORD;
	stConfig : ST_KEEL_CFG;
END_VAR
VAR
END_VAR
F_ADD_STRINGX3_TO_BUFFER( S1:= '$n#', S2:= sHead, S3:=' - Parameters:$n', wSize := wSize, pBuffer := pBuffer, wPos := wPos );

(*Targets*)
F_ADD_STRINGX4_TO_BUFFER( S1:= CONCAT(sHead, '_TgtLS_In'  ), S2:='$t', S3:= REAL_TO_STRING( stConfig.TgtLS_In  ), S4:='$n', wSize := wSize, pBuffer := pBuffer, wPos := wPos );
F_ADD_STRINGX4_TO_BUFFER( S1:= CONCAT(sHead, '_TgtLS_Mid' ), S2:='$t', S3:= REAL_TO_STRING( stConfig.TgtLS_Mid ), S4:='$n', wSize := wSize, pBuffer := pBuffer, wPos := wPos );
F_ADD_STRINGX4_TO_BUFFER( S1:= CONCAT(sHead, '_TgtLS_Out' ), S2:='$t', S3:= REAL_TO_STRING( stConfig.TgtLS_Out ), S4:='$n', wSize := wSize, pBuffer := pBuffer, wPos := wPos );

F_ADD_STRINGX4_TO_BUFFER( S1:= CONCAT(sHead, '_TgtLS_Safe_In'  ), S2:='$t', S3:= REAL_TO_STRING( stConfig.TgtLS_Safe_In  ), S4:='$n', wSize := wSize, pBuffer := pBuffer, wPos := wPos );
F_ADD_STRINGX4_TO_BUFFER( S1:= CONCAT(sHead, '_TgtLS_Safe_Out' ), S2:='$t', S3:= REAL_TO_STRING( stConfig.TgtLS_Safe_Out ), S4:='$n', wSize := wSize, pBuffer := pBuffer, wPos := wPos );

F_ADD_STRINGX4_TO_BUFFER( S1:= CONCAT(sHead, '_TgtLS_Tack_Off' ), S2:='$t', S3:= REAL_TO_STRING( stConfig.TgtLS_Tack_Off ), S4:='$n', wSize := wSize, pBuffer := pBuffer, wPos := wPos );

F_ADD_STRINGX4_TO_BUFFER( S1:= CONCAT(sHead, '_LS_DB'), S2:='$t', S3:= REAL_TO_STRING( stConfig.LS_DB ), S4:='$n', wSize := wSize, pBuffer := pBuffer, wPos := wPos );

(*Board Limits*)
F_ADD_STRINGX4_TO_BUFFER( S1:= CONCAT(sHead, '_Board_P_Min_Out'), S2:='$t', S3:= REAL_TO_STRING( stConfig.Board_P_Min_Out ), S4:='$n', wSize := wSize, pBuffer := pBuffer, wPos := wPos );
F_ADD_STRINGX4_TO_BUFFER( S1:= CONCAT(sHead, '_Board_S_Min_Out'), S2:='$t', S3:= REAL_TO_STRING( stConfig.Board_S_Min_Out ), S4:='$n', wSize := wSize, pBuffer := pBuffer, wPos := wPos );

(*Valve Limits*)
F_ADD_STRINGX4_TO_BUFFER( S1:= CONCAT(sHead, '_EVP_In_SE_Min' ), S2:='$t', S3:= REAL_TO_STRING( stConfig.EVP_In_SE_Min ), S4:='$n', wSize := wSize, pBuffer := pBuffer, wPos := wPos );
F_ADD_STRINGX4_TO_BUFFER( S1:= CONCAT(sHead, '_EVP_In_SE_Max' ), S2:='$t', S3:= REAL_TO_STRING( stConfig.EVP_In_SE_Max ), S4:='$n', wSize := wSize, pBuffer := pBuffer, wPos := wPos );
F_ADD_STRINGX4_TO_BUFFER( S1:= CONCAT(sHead, '_EVP_In_SE_Man' ), S2:='$t', S3:= REAL_TO_STRING( stConfig.EVP_In_SE_Man ), S4:='$n', wSize := wSize, pBuffer := pBuffer, wPos := wPos );

F_ADD_STRINGX4_TO_BUFFER( S1:= CONCAT(sHead, '_EVP_In_FE_Min' ), S2:='$t', S3:= REAL_TO_STRING( stConfig.EVP_In_FE_Min ), S4:='$n', wSize := wSize, pBuffer := pBuffer, wPos := wPos );
F_ADD_STRINGX4_TO_BUFFER( S1:= CONCAT(sHead, '_EVP_In_FE_Max' ), S2:='$t', S3:= REAL_TO_STRING( stConfig.EVP_In_FE_Max ), S4:='$n', wSize := wSize, pBuffer := pBuffer, wPos := wPos );
F_ADD_STRINGX4_TO_BUFFER( S1:= CONCAT(sHead, '_EVP_In_FE_Man' ), S2:='$t', S3:= REAL_TO_STRING( stConfig.EVP_In_FE_Man ), S4:='$n', wSize := wSize, pBuffer := pBuffer, wPos := wPos );

F_ADD_STRINGX4_TO_BUFFER( S1:= CONCAT(sHead, '_EVP_In_Eng_Min' ), S2:='$t', S3:= REAL_TO_STRING( stConfig.EVP_In_Eng_Min ), S4:='$n', wSize := wSize, pBuffer := pBuffer, wPos := wPos );
F_ADD_STRINGX4_TO_BUFFER( S1:= CONCAT(sHead, '_EVP_In_Eng_Max' ), S2:='$t', S3:= REAL_TO_STRING( stConfig.EVP_In_Eng_Max ), S4:='$n', wSize := wSize, pBuffer := pBuffer, wPos := wPos );
F_ADD_STRINGX4_TO_BUFFER( S1:= CONCAT(sHead, '_EVP_In_Eng_Man' ), S2:='$t', S3:= REAL_TO_STRING( stConfig.EVP_In_Eng_Man ), S4:='$n', wSize := wSize, pBuffer := pBuffer, wPos := wPos );

F_ADD_STRINGX4_TO_BUFFER( S1:= CONCAT(sHead, '_EVP_In_P_Empty' ), S2:='$t', S3:= REAL_TO_STRING( stConfig.EVP_In_P_Empty ), S4:='$n', wSize := wSize, pBuffer := pBuffer, wPos := wPos );

F_ADD_STRINGX4_TO_BUFFER( S1:= CONCAT(sHead, '_EVP_Out_SE_Min' ), S2:='$t', S3:= REAL_TO_STRING( stConfig.EVP_Out_SE_Min ), S4:='$n', wSize := wSize, pBuffer := pBuffer, wPos := wPos );
F_ADD_STRINGX4_TO_BUFFER( S1:= CONCAT(sHead, '_EVP_Out_SE_Max' ), S2:='$t', S3:= REAL_TO_STRING( stConfig.EVP_Out_SE_Max ), S4:='$n', wSize := wSize, pBuffer := pBuffer, wPos := wPos );
F_ADD_STRINGX4_TO_BUFFER( S1:= CONCAT(sHead, '_EVP_Out_SE_Man' ), S2:='$t', S3:= REAL_TO_STRING( stConfig.EVP_Out_SE_Man ), S4:='$n', wSize := wSize, pBuffer := pBuffer, wPos := wPos );
F_ADD_STRINGX4_TO_BUFFER( S1:= CONCAT(sHead, '_EVP_Out_SE_Empty' ), S2:='$t', S3:= REAL_TO_STRING( stConfig.EVP_Out_SE_Empty ), S4:='$n', wSize := wSize, pBuffer := pBuffer, wPos := wPos );

F_ADD_STRINGX4_TO_BUFFER( S1:= CONCAT(sHead, '_EVP_Out_FE_Min' ), S2:='$t', S3:= REAL_TO_STRING( stConfig.EVP_Out_FE_Min ), S4:='$n', wSize := wSize, pBuffer := pBuffer, wPos := wPos );
F_ADD_STRINGX4_TO_BUFFER( S1:= CONCAT(sHead, '_EVP_Out_FE_Max' ), S2:='$t', S3:= REAL_TO_STRING( stConfig.EVP_Out_FE_Max ), S4:='$n', wSize := wSize, pBuffer := pBuffer, wPos := wPos );
F_ADD_STRINGX4_TO_BUFFER( S1:= CONCAT(sHead, '_EVP_Out_FE_Man' ), S2:='$t', S3:= REAL_TO_STRING( stConfig.EVP_Out_FE_Man ), S4:='$n', wSize := wSize, pBuffer := pBuffer, wPos := wPos );

F_ADD_STRINGX4_TO_BUFFER( S1:= CONCAT(sHead, '_EVP_Out_Eng_Min' ), S2:='$t', S3:= REAL_TO_STRING( stConfig.EVP_Out_Eng_Min ), S4:='$n', wSize := wSize, pBuffer := pBuffer, wPos := wPos );
F_ADD_STRINGX4_TO_BUFFER( S1:= CONCAT(sHead, '_EVP_Out_Eng_Max' ), S2:='$t', S3:= REAL_TO_STRING( stConfig.EVP_Out_Eng_Max ), S4:='$n', wSize := wSize, pBuffer := pBuffer, wPos := wPos );
F_ADD_STRINGX4_TO_BUFFER( S1:= CONCAT(sHead, '_EVP_Out_Eng_Man' ), S2:='$t', S3:= REAL_TO_STRING( stConfig.EVP_Out_Eng_Man ), S4:='$n', wSize := wSize, pBuffer := pBuffer, wPos := wPos );

F_ADD_STRINGX4_TO_BUFFER( S1:= CONCAT(sHead, '_EVP_Out_Fill_Min' ), S2:='$t', S3:= REAL_TO_STRING( stConfig.EVP_Out_Fill_Min ), S4:='$n', wSize := wSize, pBuffer := pBuffer, wPos := wPos );
F_ADD_STRINGX4_TO_BUFFER( S1:= CONCAT(sHead, '_EVP_Out_Fill_Max' ), S2:='$t', S3:= REAL_TO_STRING( stConfig.EVP_Out_Fill_Max ), S4:='$n', wSize := wSize, pBuffer := pBuffer, wPos := wPos );

F_ADD_STRINGX4_TO_BUFFER( S1:= CONCAT(sHead, '_EVP_Out_P_Fill' ), S2:='$t', S3:= REAL_TO_STRING( stConfig.EVP_Out_P_Fill ), S4:='$n', wSize := wSize, pBuffer := pBuffer, wPos := wPos );

(*Valve Softstart*)

F_ADD_STRINGX4_TO_BUFFER( S1:= CONCAT(sHead, '_EVP_In_SE_Inc' ), S2:='$t', S3:= REAL_TO_STRING( stConfig.EVP_In_SE_Inc ), S4:='$n', wSize := wSize, pBuffer := pBuffer, wPos := wPos );
F_ADD_STRINGX4_TO_BUFFER( S1:= CONCAT(sHead, '_EVP_In_SE_Dec' ), S2:='$t', S3:= REAL_TO_STRING( stConfig.EVP_In_SE_Dec ), S4:='$n', wSize := wSize, pBuffer := pBuffer, wPos := wPos );

F_ADD_STRINGX4_TO_BUFFER( S1:= CONCAT(sHead, '_EVP_In_FE_Inc' ), S2:='$t', S3:= REAL_TO_STRING( stConfig.EVP_In_FE_Inc ), S4:='$n', wSize := wSize, pBuffer := pBuffer, wPos := wPos );
F_ADD_STRINGX4_TO_BUFFER( S1:= CONCAT(sHead, '_EVP_In_FE_Dec' ), S2:='$t', S3:= REAL_TO_STRING( stConfig.EVP_In_FE_Dec ), S4:='$n', wSize := wSize, pBuffer := pBuffer, wPos := wPos );

F_ADD_STRINGX4_TO_BUFFER( S1:= CONCAT(sHead, '_EVP_Out_SE_Inc' ), S2:='$t', S3:= REAL_TO_STRING( stConfig.EVP_Out_SE_Inc ), S4:='$n', wSize := wSize, pBuffer := pBuffer, wPos := wPos );
F_ADD_STRINGX4_TO_BUFFER( S1:= CONCAT(sHead, '_EVP_Out_SE_Dec' ), S2:='$t', S3:= REAL_TO_STRING( stConfig.EVP_Out_SE_Dec ), S4:='$n', wSize := wSize, pBuffer := pBuffer, wPos := wPos );

F_ADD_STRINGX4_TO_BUFFER( S1:= CONCAT(sHead, '_EVP_Out_FE_Inc' ), S2:='$t', S3:= REAL_TO_STRING( stConfig.EVP_Out_FE_Inc ), S4:='$n', wSize := wSize, pBuffer := pBuffer, wPos := wPos );
F_ADD_STRINGX4_TO_BUFFER( S1:= CONCAT(sHead, '_EVP_Out_FE_Dec' ), S2:='$t', S3:= REAL_TO_STRING( stConfig.EVP_Out_FE_Dec ), S4:='$n', wSize := wSize, pBuffer := pBuffer, wPos := wPos );

F_ADD_STRINGX4_TO_BUFFER( S1:= CONCAT(sHead, '_EVP_In_Eng_Inc' ), S2:='$t', S3:= REAL_TO_STRING( stConfig.EVP_In_Eng_Inc ), S4:='$n', wSize := wSize, pBuffer := pBuffer, wPos := wPos );
F_ADD_STRINGX4_TO_BUFFER( S1:= CONCAT(sHead, '_EVP_In_Eng_Dec' ), S2:='$t', S3:= REAL_TO_STRING( stConfig.EVP_In_Eng_Dec ), S4:='$n', wSize := wSize, pBuffer := pBuffer, wPos := wPos );

F_ADD_STRINGX4_TO_BUFFER( S1:= CONCAT(sHead, '_EVP_Out_Eng_Inc' ), S2:='$t', S3:= REAL_TO_STRING( stConfig.EVP_Out_Eng_Inc ), S4:='$n', wSize := wSize, pBuffer := pBuffer, wPos := wPos );
F_ADD_STRINGX4_TO_BUFFER( S1:= CONCAT(sHead, '_EVP_Out_Eng_Dec' ), S2:='$t', S3:= REAL_TO_STRING( stConfig.EVP_Out_Eng_Dec ), S4:='$n', wSize := wSize, pBuffer := pBuffer, wPos := wPos );

(*Valve Gains*)
F_ADD_STRINGX4_TO_BUFFER( S1:= CONCAT(sHead, '_EVP_In_Eng_K'  ), S2:='$t', S3:= REAL_TO_STRING( stConfig.EVP_In_Eng_K  ), S4:='$n', wSize := wSize, pBuffer := pBuffer, wPos := wPos );
F_ADD_STRINGX4_TO_BUFFER( S1:= CONCAT(sHead, '_EVP_Out_Eng_K' ), S2:='$t', S3:= REAL_TO_STRING( stConfig.EVP_Out_Eng_K ), S4:='$n', wSize := wSize, pBuffer := pBuffer, wPos := wPos );

F_ADD_STRINGX4_TO_BUFFER( S1:= CONCAT(sHead, '_LP'  ), S2:='$t', S3:= BYTE_TO_STRING( stConfig.LP ), S4:='$n', wSize := wSize, pBuffer := pBuffer, wPos := wPos );

F_ADD_STRINGX4_TO_BUFFER( S1:= CONCAT(sHead, '_TimeMax'  ), S2:='$t', S3:= REAL_TO_STRING( stConfig.TimeMax  ), S4:='$n', wSize := wSize, pBuffer := pBuffer, wPos := wPos );

(*Auto Ease limit*)
F_ADD_STRINGX4_TO_BUFFER( S1:= CONCAT(sHead, '_MinLoadSide_Bar'   ), S2:='$t', S3:= REAL_TO_STRING( stConfig.MinLoadSide_Bar   ), S4:='$n', wSize := wSize, pBuffer := pBuffer, wPos := wPos );
F_ADD_STRINGX4_TO_BUFFER( S1:= CONCAT(sHead, '_MaxUnloadSide_Bar' ), S2:='$t', S3:= REAL_TO_STRING( stConfig.MaxUnloadSide_Bar ), S4:='$n', wSize := wSize, pBuffer := pBuffer, wPos := wPos );
END_FUNCTION

(* POU FUN/PARAMETERS/F_WRITE_TRAVELLER_CFG, ST *)
FUNCTION F_WRITE_TRAVELLER_CFG : BOOL
VAR_INPUT
	sHead : STRING;
	wSize   :DWORD;
	pBuffer :POINTER TO BYTE;
END_VAR
VAR_IN_OUT
	wPos     : DWORD;
	stConfig : ST_TRAVELLER_CFG;
END_VAR
VAR
END_VAR
F_ADD_STRINGX3_TO_BUFFER( S1:= '$n#', S2:= sHead, S3:=' - Parameters:$n', wSize := wSize, pBuffer := pBuffer, wPos := wPos );

F_ADD_STRINGX4_TO_BUFFER( S1:= CONCAT(sHead, '_MaxEVPA' ), S2:='$t', S3:= REAL_TO_STRING( stConfig.MaxEVPA ), S4:='$n', wSize := wSize, pBuffer := pBuffer, wPos := wPos );
F_ADD_STRINGX4_TO_BUFFER( S1:= CONCAT(sHead, '_MaxEVPB' ), S2:='$t', S3:= REAL_TO_STRING( stConfig.MaxEVPB ), S4:='$n', wSize := wSize, pBuffer := pBuffer, wPos := wPos );
F_ADD_STRINGX4_TO_BUFFER( S1:= CONCAT(sHead, '_MinEVPA' ), S2:='$t', S3:= REAL_TO_STRING( stConfig.MinEVPA ), S4:='$n', wSize := wSize, pBuffer := pBuffer, wPos := wPos );
F_ADD_STRINGX4_TO_BUFFER( S1:= CONCAT(sHead, '_MinEVPB' ), S2:='$t', S3:= REAL_TO_STRING( stConfig.MinEVPB ), S4:='$n', wSize := wSize, pBuffer := pBuffer, wPos := wPos );

F_ADD_STRINGX4_TO_BUFFER( S1:= CONCAT(sHead, '_Spd_Inc' ), S2:='$t', S3:= REAL_TO_STRING( stConfig.Spd_Inc ), S4:='$n', wSize := wSize, pBuffer := pBuffer, wPos := wPos );
F_ADD_STRINGX4_TO_BUFFER( S1:= CONCAT(sHead, '_Spd_Dec' ), S2:='$t', S3:= REAL_TO_STRING( stConfig.Spd_Dec ), S4:='$n', wSize := wSize, pBuffer := pBuffer, wPos := wPos );

F_ADD_STRINGX4_TO_BUFFER( S1:= CONCAT(sHead, '_TgtLS_Max'  ), S2:='$t', S3:= REAL_TO_STRING( stConfig.TgtLS_Max  ), S4:='$n', wSize := wSize, pBuffer := pBuffer, wPos := wPos );
F_ADD_STRINGX4_TO_BUFFER( S1:= CONCAT(sHead, '_TgtLS_Zero' ), S2:='$t', S3:= REAL_TO_STRING( stConfig.TgtLS_Zero ), S4:='$n', wSize := wSize, pBuffer := pBuffer, wPos := wPos );
F_ADD_STRINGX4_TO_BUFFER( S1:= CONCAT(sHead, '_TgtLS_Min'  ), S2:='$t', S3:= REAL_TO_STRING( stConfig.TgtLS_Min  ), S4:='$n', wSize := wSize, pBuffer := pBuffer, wPos := wPos );

F_ADD_STRINGX4_TO_BUFFER( S1:= CONCAT(sHead, '_TgtLS_Tack_Off' ), S2:='$t', S3:= REAL_TO_STRING( stConfig.TgtLS_Tack_Off ), S4:='$n', wSize := wSize, pBuffer := pBuffer, wPos := wPos );

F_ADD_STRINGX4_TO_BUFFER( S1:= CONCAT(sHead, '_LS_DB'    ), S2:='$t', S3:= REAL_TO_STRING( stConfig.LS_DB    ), S4:='$n', wSize := wSize, pBuffer := pBuffer, wPos := wPos );
F_ADD_STRINGX4_TO_BUFFER( S1:= CONCAT(sHead, '_LS_Dist'  ), S2:='$t', S3:= REAL_TO_STRING( stConfig.LS_Dist  ), S4:='$n', wSize := wSize, pBuffer := pBuffer, wPos := wPos );
F_ADD_STRINGX4_TO_BUFFER( S1:= CONCAT(sHead, '_LS_Limit' ), S2:='$t', S3:= BOOL_TO_STRING( stConfig.LS_Limit ), S4:='$n', wSize := wSize, pBuffer := pBuffer, wPos := wPos );

F_ADD_STRINGX4_TO_BUFFER( S1:= CONCAT(sHead, '_TimeMax'  ), S2:='$t', S3:= REAL_TO_STRING( stConfig.TimeMax  ), S4:='$n', wSize := wSize, pBuffer := pBuffer, wPos := wPos );

F_ADD_STRINGX4_TO_BUFFER( S1:= CONCAT(sHead, '_Hyst_HP' ), S2:='$t', S3:= REAL_TO_STRING( stConfig.Hyst_HP ), S4:='$n', wSize := wSize, pBuffer := pBuffer, wPos := wPos );
F_ADD_STRINGX4_TO_BUFFER( S1:= CONCAT(sHead, '_Hyst_LP' ), S2:='$t', S3:= REAL_TO_STRING( stConfig.Hyst_LP ), S4:='$n', wSize := wSize, pBuffer := pBuffer, wPos := wPos );
F_ADD_STRINGX4_TO_BUFFER( S1:= CONCAT(sHead, '_Hyst_TM' ), S2:='$t', S3:= REAL_TO_STRING( stConfig.Hyst_TM ), S4:='$n', wSize := wSize, pBuffer := pBuffer, wPos := wPos );

F_ADD_STRINGX4_TO_BUFFER( S1:= CONCAT(sHead, '_HP'  ), S2:='$t', S3:= BYTE_TO_STRING( stConfig.HP ), S4:='$n', wSize := wSize, pBuffer := pBuffer, wPos := wPos );
F_ADD_STRINGX4_TO_BUFFER( S1:= CONCAT(sHead, '_LP'  ), S2:='$t', S3:= BYTE_TO_STRING( stConfig.LP ), S4:='$n', wSize := wSize, pBuffer := pBuffer, wPos := wPos );
END_FUNCTION

(* POU FUN/PARAMETERS/F_WRITE_LP_FUNC_CFG, ST *)
FUNCTION F_WRITE_LP_FUNC_CFG : BOOL
VAR_INPUT
	sHead : STRING;
	wSize   :DWORD;
	pBuffer :POINTER TO BYTE;
END_VAR
VAR_IN_OUT
	wPos     : DWORD;
	stConfig : ST_LP_FUNC_CFG;
END_VAR
VAR

END_VAR
F_ADD_STRINGX3_TO_BUFFER( S1:= '$n#', S2:= sHead, S3:=' - Parameters:$n', wSize := wSize, pBuffer := pBuffer, wPos := wPos );

F_ADD_STRINGX4_TO_BUFFER( S1:= CONCAT(sHead, '_SpdA_Min' ), S2:='$t', S3:= REAL_TO_STRING( stConfig.SpdA_Min ), S4:='$n', wSize := wSize, pBuffer := pBuffer, wPos := wPos );
F_ADD_STRINGX4_TO_BUFFER( S1:= CONCAT(sHead, '_SpdA_Max' ), S2:='$t', S3:= REAL_TO_STRING( stConfig.SpdA_Max ), S4:='$n', wSize := wSize, pBuffer := pBuffer, wPos := wPos );
F_ADD_STRINGX4_TO_BUFFER( S1:= CONCAT(sHead, '_SpdB_Min' ), S2:='$t', S3:= REAL_TO_STRING( stConfig.SpdB_Min ), S4:='$n', wSize := wSize, pBuffer := pBuffer, wPos := wPos );
F_ADD_STRINGX4_TO_BUFFER( S1:= CONCAT(sHead, '_SpdB_Max' ), S2:='$t', S3:= REAL_TO_STRING( stConfig.SpdB_MAx ), S4:='$n', wSize := wSize, pBuffer := pBuffer, wPos := wPos );

F_ADD_STRINGX4_TO_BUFFER( S1:= CONCAT(sHead, '_Spd_Inc' ), S2:='$t', S3:= REAL_TO_STRING( stConfig.Spd_Inc ), S4:='$n', wSize := wSize, pBuffer := pBuffer, wPos := wPos );
F_ADD_STRINGX4_TO_BUFFER( S1:= CONCAT(sHead, '_Spd_Dec' ), S2:='$t', S3:= REAL_TO_STRING( stConfig.Spd_Dec ), S4:='$n', wSize := wSize, pBuffer := pBuffer, wPos := wPos );

F_ADD_STRINGX4_TO_BUFFER( S1:= CONCAT(sHead, '_SF1_Limit' ), S2:='$t', S3:= BOOL_TO_STRING( stConfig.SF1_Limit ), S4:='$n', wSize := wSize, pBuffer := pBuffer, wPos := wPos );
F_ADD_STRINGX4_TO_BUFFER( S1:= CONCAT(sHead, '_SF2_Limit' ), S2:='$t', S3:= BOOL_TO_STRING( stConfig.SF2_Limit ), S4:='$n', wSize := wSize, pBuffer := pBuffer, wPos := wPos );

F_ADD_STRINGX4_TO_BUFFER( S1:= CONCAT(sHead, '_A_Spd1' ), S2:='$t', S3:= BOOL_TO_STRING( stConfig.A_Spd1 ), S4:='$n', wSize := wSize, pBuffer := pBuffer, wPos := wPos );

F_ADD_STRINGX4_TO_BUFFER( S1:= CONCAT(sHead, '_TimeMax' ), S2:='$t', S3:= REAL_TO_STRING( stConfig.TimeMax ), S4:='$n', wSize := wSize, pBuffer := pBuffer, wPos := wPos );
END_FUNCTION

(* POU FUN/PARAMETERS/F_WRITE_TACK_VALVE_CFG, ST *)
FUNCTION F_WRITE_TACK_VALVE_CFG : BOOL
VAR_INPUT
	sHead : STRING;
	wSize   :DWORD;
	pBuffer :POINTER TO BYTE;
END_VAR
VAR_IN_OUT
	wPos     : DWORD;
	stConfig : ST_TACK_VALVE_CFG;
END_VAR
VAR
END_VAR
F_ADD_STRINGX3_TO_BUFFER( S1:= '$n#', S2:= sHead, S3:=' - Parameters:$n', wSize := wSize, pBuffer := pBuffer, wPos := wPos );

F_ADD_STRINGX4_TO_BUFFER( S1:= CONCAT(sHead, '_TimeMax'   ), S2:='$t', S3:= REAL_TO_STRING( stConfig.TimeMax  ), S4:='$n', wSize := wSize, pBuffer := pBuffer, wPos := wPos );

F_ADD_STRINGX4_TO_BUFFER( S1:= CONCAT(sHead, '_Hyst_HeelH' ), S2:='$t', S3:= REAL_TO_STRING( stConfig.Hyst_HeelH ), S4:='$n', wSize := wSize, pBuffer := pBuffer, wPos := wPos );
F_ADD_STRINGX4_TO_BUFFER( S1:= CONCAT(sHead, '_Hyst_HeelL' ), S2:='$t', S3:= REAL_TO_STRING( stConfig.Hyst_HeelL ), S4:='$n', wSize := wSize, pBuffer := pBuffer, wPos := wPos );
F_ADD_STRINGX4_TO_BUFFER( S1:= CONCAT(sHead, '_Hyst_Time'  ), S2:='$t', S3:= REAL_TO_STRING( stConfig.Hyst_Time  ), S4:='$n', wSize := wSize, pBuffer := pBuffer, wPos := wPos );
END_FUNCTION

(* POU FUN/PARAMETERS/F_WRITE_MAST_SETUP_CFG, ST *)
FUNCTION F_WRITE_MAST_SETUP_CFG : BOOL
VAR_INPUT
	sHead : STRING;
	wSize   :DWORD;
	pBuffer :POINTER TO BYTE;
END_VAR
VAR_IN_OUT
	wPos     : DWORD;
	stTABLE : ST_MAST_SETUP;
END_VAR
VAR
END_VAR
F_ADD_STRINGX3_TO_BUFFER( S1:= '$n#', S2:= sHead, S3:=' - Parameters:$n', wSize := wSize, pBuffer := pBuffer, wPos := wPos );

F_ADD_STRINGX4_TO_BUFFER( S1:= CONCAT(sHead, '_FSY_1_1' ), S2:='$t', S3:= REAL_TO_STRING( stTABLE.aFSY[1,1] ), S4:='$n', wSize := wSize, pBuffer := pBuffer, wPos := wPos );
F_ADD_STRINGX4_TO_BUFFER( S1:= CONCAT(sHead, '_FSY_1_2' ), S2:='$t', S3:= REAL_TO_STRING( stTABLE.aFSY[1,2] ), S4:='$n', wSize := wSize, pBuffer := pBuffer, wPos := wPos );
F_ADD_STRINGX4_TO_BUFFER( S1:= CONCAT(sHead, '_FSY_1_3' ), S2:='$t', S3:= REAL_TO_STRING( stTABLE.aFSY[1,3] ), S4:='$n', wSize := wSize, pBuffer := pBuffer, wPos := wPos );
F_ADD_STRINGX4_TO_BUFFER( S1:= CONCAT(sHead, '_FSY_1_4' ), S2:='$t', S3:= REAL_TO_STRING( stTABLE.aFSY[1,4] ), S4:='$n', wSize := wSize, pBuffer := pBuffer, wPos := wPos );
F_ADD_STRINGX4_TO_BUFFER( S1:= CONCAT(sHead, '_FSY_1_5' ), S2:='$t', S3:= REAL_TO_STRING( stTABLE.aFSY[1,5] ), S4:='$n', wSize := wSize, pBuffer := pBuffer, wPos := wPos );
F_ADD_STRINGX4_TO_BUFFER( S1:= CONCAT(sHead, '_FSY_1_6' ), S2:='$t', S3:= REAL_TO_STRING( stTABLE.aFSY[1,6] ), S4:='$n', wSize := wSize, pBuffer := pBuffer, wPos := wPos );

F_ADD_STRINGX4_TO_BUFFER( S1:= CONCAT(sHead, '_FSY_2_1' ), S2:='$t', S3:= REAL_TO_STRING( stTABLE.aFSY[2,1] ), S4:='$n', wSize := wSize, pBuffer := pBuffer, wPos := wPos );
F_ADD_STRINGX4_TO_BUFFER( S1:= CONCAT(sHead, '_FSY_2_2' ), S2:='$t', S3:= REAL_TO_STRING( stTABLE.aFSY[2,2] ), S4:='$n', wSize := wSize, pBuffer := pBuffer, wPos := wPos );
F_ADD_STRINGX4_TO_BUFFER( S1:= CONCAT(sHead, '_FSY_2_3' ), S2:='$t', S3:= REAL_TO_STRING( stTABLE.aFSY[2,3] ), S4:='$n', wSize := wSize, pBuffer := pBuffer, wPos := wPos );
F_ADD_STRINGX4_TO_BUFFER( S1:= CONCAT(sHead, '_FSY_2_4' ), S2:='$t', S3:= REAL_TO_STRING( stTABLE.aFSY[2,4] ), S4:='$n', wSize := wSize, pBuffer := pBuffer, wPos := wPos );
F_ADD_STRINGX4_TO_BUFFER( S1:= CONCAT(sHead, '_FSY_2_5' ), S2:='$t', S3:= REAL_TO_STRING( stTABLE.aFSY[2,5] ), S4:='$n', wSize := wSize, pBuffer := pBuffer, wPos := wPos );
F_ADD_STRINGX4_TO_BUFFER( S1:= CONCAT(sHead, '_FSY_2_6' ), S2:='$t', S3:= REAL_TO_STRING( stTABLE.aFSY[2,6] ), S4:='$n', wSize := wSize, pBuffer := pBuffer, wPos := wPos );

F_ADD_STRINGX4_TO_BUFFER( S1:= CONCAT(sHead, '_FSY_3_1' ), S2:='$t', S3:= REAL_TO_STRING( stTABLE.aFSY[3,1] ), S4:='$n', wSize := wSize, pBuffer := pBuffer, wPos := wPos );
F_ADD_STRINGX4_TO_BUFFER( S1:= CONCAT(sHead, '_FSY_3_2' ), S2:='$t', S3:= REAL_TO_STRING( stTABLE.aFSY[3,2] ), S4:='$n', wSize := wSize, pBuffer := pBuffer, wPos := wPos );
F_ADD_STRINGX4_TO_BUFFER( S1:= CONCAT(sHead, '_FSY_3_3' ), S2:='$t', S3:= REAL_TO_STRING( stTABLE.aFSY[3,3] ), S4:='$n', wSize := wSize, pBuffer := pBuffer, wPos := wPos );
F_ADD_STRINGX4_TO_BUFFER( S1:= CONCAT(sHead, '_FSY_3_4' ), S2:='$t', S3:= REAL_TO_STRING( stTABLE.aFSY[3,4] ), S4:='$n', wSize := wSize, pBuffer := pBuffer, wPos := wPos );
F_ADD_STRINGX4_TO_BUFFER( S1:= CONCAT(sHead, '_FSY_3_5' ), S2:='$t', S3:= REAL_TO_STRING( stTABLE.aFSY[3,5] ), S4:='$n', wSize := wSize, pBuffer := pBuffer, wPos := wPos );
F_ADD_STRINGX4_TO_BUFFER( S1:= CONCAT(sHead, '_FSY_3_6' ), S2:='$t', S3:= REAL_TO_STRING( stTABLE.aFSY[3,6] ), S4:='$n', wSize := wSize, pBuffer := pBuffer, wPos := wPos );

F_ADD_STRINGX4_TO_BUFFER( S1:= CONCAT(sHead, '_FSY_4_1' ), S2:='$t', S3:= REAL_TO_STRING( stTABLE.aFSY[4,1] ), S4:='$n', wSize := wSize, pBuffer := pBuffer, wPos := wPos );
F_ADD_STRINGX4_TO_BUFFER( S1:= CONCAT(sHead, '_FSY_4_2' ), S2:='$t', S3:= REAL_TO_STRING( stTABLE.aFSY[4,2] ), S4:='$n', wSize := wSize, pBuffer := pBuffer, wPos := wPos );
F_ADD_STRINGX4_TO_BUFFER( S1:= CONCAT(sHead, '_FSY_4_3' ), S2:='$t', S3:= REAL_TO_STRING( stTABLE.aFSY[4,3] ), S4:='$n', wSize := wSize, pBuffer := pBuffer, wPos := wPos );
F_ADD_STRINGX4_TO_BUFFER( S1:= CONCAT(sHead, '_FSY_4_4' ), S2:='$t', S3:= REAL_TO_STRING( stTABLE.aFSY[4,4] ), S4:='$n', wSize := wSize, pBuffer := pBuffer, wPos := wPos );
F_ADD_STRINGX4_TO_BUFFER( S1:= CONCAT(sHead, '_FSY_4_5' ), S2:='$t', S3:= REAL_TO_STRING( stTABLE.aFSY[4,5] ), S4:='$n', wSize := wSize, pBuffer := pBuffer, wPos := wPos );
F_ADD_STRINGX4_TO_BUFFER( S1:= CONCAT(sHead, '_FSY_4_6' ), S2:='$t', S3:= REAL_TO_STRING( stTABLE.aFSY[4,6] ), S4:='$n', wSize := wSize, pBuffer := pBuffer, wPos := wPos );

F_ADD_STRINGX4_TO_BUFFER( S1:= CONCAT(sHead, '_BDEF_1_1' ), S2:='$t', S3:= REAL_TO_STRING( stTABLE.aBDef[1,1] ), S4:='$n', wSize := wSize, pBuffer := pBuffer, wPos := wPos );
F_ADD_STRINGX4_TO_BUFFER( S1:= CONCAT(sHead, '_BDEF_1_2' ), S2:='$t', S3:= REAL_TO_STRING( stTABLE.aBDef[1,2] ), S4:='$n', wSize := wSize, pBuffer := pBuffer, wPos := wPos );
F_ADD_STRINGX4_TO_BUFFER( S1:= CONCAT(sHead, '_BDEF_1_3' ), S2:='$t', S3:= REAL_TO_STRING( stTABLE.aBDef[1,3] ), S4:='$n', wSize := wSize, pBuffer := pBuffer, wPos := wPos );
F_ADD_STRINGX4_TO_BUFFER( S1:= CONCAT(sHead, '_BDEF_1_4' ), S2:='$t', S3:= REAL_TO_STRING( stTABLE.aBDef[1,4] ), S4:='$n', wSize := wSize, pBuffer := pBuffer, wPos := wPos );
F_ADD_STRINGX4_TO_BUFFER( S1:= CONCAT(sHead, '_BDEF_1_5' ), S2:='$t', S3:= REAL_TO_STRING( stTABLE.aBDef[1,5] ), S4:='$n', wSize := wSize, pBuffer := pBuffer, wPos := wPos );
F_ADD_STRINGX4_TO_BUFFER( S1:= CONCAT(sHead, '_BDEF_1_6' ), S2:='$t', S3:= REAL_TO_STRING( stTABLE.aBDef[1,6] ), S4:='$n', wSize := wSize, pBuffer := pBuffer, wPos := wPos );

F_ADD_STRINGX4_TO_BUFFER( S1:= CONCAT(sHead, '_BDEF_2_1' ), S2:='$t', S3:= REAL_TO_STRING( stTABLE.aBDef[2,1] ), S4:='$n', wSize := wSize, pBuffer := pBuffer, wPos := wPos );
F_ADD_STRINGX4_TO_BUFFER( S1:= CONCAT(sHead, '_BDEF_2_2' ), S2:='$t', S3:= REAL_TO_STRING( stTABLE.aBDef[2,2] ), S4:='$n', wSize := wSize, pBuffer := pBuffer, wPos := wPos );
F_ADD_STRINGX4_TO_BUFFER( S1:= CONCAT(sHead, '_BDEF_2_3' ), S2:='$t', S3:= REAL_TO_STRING( stTABLE.aBDef[2,3] ), S4:='$n', wSize := wSize, pBuffer := pBuffer, wPos := wPos );
F_ADD_STRINGX4_TO_BUFFER( S1:= CONCAT(sHead, '_BDEF_2_4' ), S2:='$t', S3:= REAL_TO_STRING( stTABLE.aBDef[2,4] ), S4:='$n', wSize := wSize, pBuffer := pBuffer, wPos := wPos );
F_ADD_STRINGX4_TO_BUFFER( S1:= CONCAT(sHead, '_BDEF_2_5' ), S2:='$t', S3:= REAL_TO_STRING( stTABLE.aBDef[2,5] ), S4:='$n', wSize := wSize, pBuffer := pBuffer, wPos := wPos );
F_ADD_STRINGX4_TO_BUFFER( S1:= CONCAT(sHead, '_BDEF_2_6' ), S2:='$t', S3:= REAL_TO_STRING( stTABLE.aBDef[2,6] ), S4:='$n', wSize := wSize, pBuffer := pBuffer, wPos := wPos );

F_ADD_STRINGX4_TO_BUFFER( S1:= CONCAT(sHead, '_BDEF_3_1' ), S2:='$t', S3:= REAL_TO_STRING( stTABLE.aBDef[3,1] ), S4:='$n', wSize := wSize, pBuffer := pBuffer, wPos := wPos );
F_ADD_STRINGX4_TO_BUFFER( S1:= CONCAT(sHead, '_BDEF_3_2' ), S2:='$t', S3:= REAL_TO_STRING( stTABLE.aBDef[3,2] ), S4:='$n', wSize := wSize, pBuffer := pBuffer, wPos := wPos );
F_ADD_STRINGX4_TO_BUFFER( S1:= CONCAT(sHead, '_BDEF_3_3' ), S2:='$t', S3:= REAL_TO_STRING( stTABLE.aBDef[3,3] ), S4:='$n', wSize := wSize, pBuffer := pBuffer, wPos := wPos );
F_ADD_STRINGX4_TO_BUFFER( S1:= CONCAT(sHead, '_BDEF_3_4' ), S2:='$t', S3:= REAL_TO_STRING( stTABLE.aBDef[3,4] ), S4:='$n', wSize := wSize, pBuffer := pBuffer, wPos := wPos );
F_ADD_STRINGX4_TO_BUFFER( S1:= CONCAT(sHead, '_BDEF_3_5' ), S2:='$t', S3:= REAL_TO_STRING( stTABLE.aBDef[3,5] ), S4:='$n', wSize := wSize, pBuffer := pBuffer, wPos := wPos );
F_ADD_STRINGX4_TO_BUFFER( S1:= CONCAT(sHead, '_BDEF_3_6' ), S2:='$t', S3:= REAL_TO_STRING( stTABLE.aBDef[3,6] ), S4:='$n', wSize := wSize, pBuffer := pBuffer, wPos := wPos );

F_ADD_STRINGX4_TO_BUFFER( S1:= CONCAT(sHead, '_BDEF_4_1' ), S2:='$t', S3:= REAL_TO_STRING( stTABLE.aBDef[4,1] ), S4:='$n', wSize := wSize, pBuffer := pBuffer, wPos := wPos );
F_ADD_STRINGX4_TO_BUFFER( S1:= CONCAT(sHead, '_BDEF_4_2' ), S2:='$t', S3:= REAL_TO_STRING( stTABLE.aBDef[4,2] ), S4:='$n', wSize := wSize, pBuffer := pBuffer, wPos := wPos );
F_ADD_STRINGX4_TO_BUFFER( S1:= CONCAT(sHead, '_BDEF_4_3' ), S2:='$t', S3:= REAL_TO_STRING( stTABLE.aBDef[4,3] ), S4:='$n', wSize := wSize, pBuffer := pBuffer, wPos := wPos );
F_ADD_STRINGX4_TO_BUFFER( S1:= CONCAT(sHead, '_BDEF_4_4' ), S2:='$t', S3:= REAL_TO_STRING( stTABLE.aBDef[4,4] ), S4:='$n', wSize := wSize, pBuffer := pBuffer, wPos := wPos );
F_ADD_STRINGX4_TO_BUFFER( S1:= CONCAT(sHead, '_BDEF_4_5' ), S2:='$t', S3:= REAL_TO_STRING( stTABLE.aBDef[4,5] ), S4:='$n', wSize := wSize, pBuffer := pBuffer, wPos := wPos );
F_ADD_STRINGX4_TO_BUFFER( S1:= CONCAT(sHead, '_BDEF_4_6' ), S2:='$t', S3:= REAL_TO_STRING( stTABLE.aBDef[4,6] ), S4:='$n', wSize := wSize, pBuffer := pBuffer, wPos := wPos );

F_ADD_STRINGX4_TO_BUFFER( S1:= CONCAT(sHead, '_TDEF_1_1' ), S2:='$t', S3:= REAL_TO_STRING( stTABLE.aTDef[1,1] ), S4:='$n', wSize := wSize, pBuffer := pBuffer, wPos := wPos );
F_ADD_STRINGX4_TO_BUFFER( S1:= CONCAT(sHead, '_TDEF_1_2' ), S2:='$t', S3:= REAL_TO_STRING( stTABLE.aTDef[1,2] ), S4:='$n', wSize := wSize, pBuffer := pBuffer, wPos := wPos );
F_ADD_STRINGX4_TO_BUFFER( S1:= CONCAT(sHead, '_TDEF_1_3' ), S2:='$t', S3:= REAL_TO_STRING( stTABLE.aTDef[1,3] ), S4:='$n', wSize := wSize, pBuffer := pBuffer, wPos := wPos );
F_ADD_STRINGX4_TO_BUFFER( S1:= CONCAT(sHead, '_TDEF_1_4' ), S2:='$t', S3:= REAL_TO_STRING( stTABLE.aTDef[1,4] ), S4:='$n', wSize := wSize, pBuffer := pBuffer, wPos := wPos );
F_ADD_STRINGX4_TO_BUFFER( S1:= CONCAT(sHead, '_TDEF_1_5' ), S2:='$t', S3:= REAL_TO_STRING( stTABLE.aTDef[1,5] ), S4:='$n', wSize := wSize, pBuffer := pBuffer, wPos := wPos );
F_ADD_STRINGX4_TO_BUFFER( S1:= CONCAT(sHead, '_TDEF_1_6' ), S2:='$t', S3:= REAL_TO_STRING( stTABLE.aTDef[1,6] ), S4:='$n', wSize := wSize, pBuffer := pBuffer, wPos := wPos );

F_ADD_STRINGX4_TO_BUFFER( S1:= CONCAT(sHead, '_TDEF_2_1' ), S2:='$t', S3:= REAL_TO_STRING( stTABLE.aTDef[2,1] ), S4:='$n', wSize := wSize, pBuffer := pBuffer, wPos := wPos );
F_ADD_STRINGX4_TO_BUFFER( S1:= CONCAT(sHead, '_TDEF_2_2' ), S2:='$t', S3:= REAL_TO_STRING( stTABLE.aTDef[2,2] ), S4:='$n', wSize := wSize, pBuffer := pBuffer, wPos := wPos );
F_ADD_STRINGX4_TO_BUFFER( S1:= CONCAT(sHead, '_TDEF_2_3' ), S2:='$t', S3:= REAL_TO_STRING( stTABLE.aTDef[2,3] ), S4:='$n', wSize := wSize, pBuffer := pBuffer, wPos := wPos );
F_ADD_STRINGX4_TO_BUFFER( S1:= CONCAT(sHead, '_TDEF_2_4' ), S2:='$t', S3:= REAL_TO_STRING( stTABLE.aTDef[2,4] ), S4:='$n', wSize := wSize, pBuffer := pBuffer, wPos := wPos );
F_ADD_STRINGX4_TO_BUFFER( S1:= CONCAT(sHead, '_TDEF_2_5' ), S2:='$t', S3:= REAL_TO_STRING( stTABLE.aTDef[2,5] ), S4:='$n', wSize := wSize, pBuffer := pBuffer, wPos := wPos );
F_ADD_STRINGX4_TO_BUFFER( S1:= CONCAT(sHead, '_TDEF_2_6' ), S2:='$t', S3:= REAL_TO_STRING( stTABLE.aTDef[2,6] ), S4:='$n', wSize := wSize, pBuffer := pBuffer, wPos := wPos );

F_ADD_STRINGX4_TO_BUFFER( S1:= CONCAT(sHead, '_TDEF_3_1' ), S2:='$t', S3:= REAL_TO_STRING( stTABLE.aTDef[3,1] ), S4:='$n', wSize := wSize, pBuffer := pBuffer, wPos := wPos );
F_ADD_STRINGX4_TO_BUFFER( S1:= CONCAT(sHead, '_TDEF_3_2' ), S2:='$t', S3:= REAL_TO_STRING( stTABLE.aTDef[3,2] ), S4:='$n', wSize := wSize, pBuffer := pBuffer, wPos := wPos );
F_ADD_STRINGX4_TO_BUFFER( S1:= CONCAT(sHead, '_TDEF_3_3' ), S2:='$t', S3:= REAL_TO_STRING( stTABLE.aTDef[3,3] ), S4:='$n', wSize := wSize, pBuffer := pBuffer, wPos := wPos );
F_ADD_STRINGX4_TO_BUFFER( S1:= CONCAT(sHead, '_TDEF_3_4' ), S2:='$t', S3:= REAL_TO_STRING( stTABLE.aTDef[3,4] ), S4:='$n', wSize := wSize, pBuffer := pBuffer, wPos := wPos );
F_ADD_STRINGX4_TO_BUFFER( S1:= CONCAT(sHead, '_TDEF_3_5' ), S2:='$t', S3:= REAL_TO_STRING( stTABLE.aTDef[3,5] ), S4:='$n', wSize := wSize, pBuffer := pBuffer, wPos := wPos );
F_ADD_STRINGX4_TO_BUFFER( S1:= CONCAT(sHead, '_TDEF_3_6' ), S2:='$t', S3:= REAL_TO_STRING( stTABLE.aTDef[3,6] ), S4:='$n', wSize := wSize, pBuffer := pBuffer, wPos := wPos );

F_ADD_STRINGX4_TO_BUFFER( S1:= CONCAT(sHead, '_TDEF_4_1' ), S2:='$t', S3:= REAL_TO_STRING( stTABLE.aTDef[4,1] ), S4:='$n', wSize := wSize, pBuffer := pBuffer, wPos := wPos );
F_ADD_STRINGX4_TO_BUFFER( S1:= CONCAT(sHead, '_TDEF_4_2' ), S2:='$t', S3:= REAL_TO_STRING( stTABLE.aTDef[4,2] ), S4:='$n', wSize := wSize, pBuffer := pBuffer, wPos := wPos );
F_ADD_STRINGX4_TO_BUFFER( S1:= CONCAT(sHead, '_TDEF_4_3' ), S2:='$t', S3:= REAL_TO_STRING( stTABLE.aTDef[4,3] ), S4:='$n', wSize := wSize, pBuffer := pBuffer, wPos := wPos );
F_ADD_STRINGX4_TO_BUFFER( S1:= CONCAT(sHead, '_TDEF_4_4' ), S2:='$t', S3:= REAL_TO_STRING( stTABLE.aTDef[4,4] ), S4:='$n', wSize := wSize, pBuffer := pBuffer, wPos := wPos );
F_ADD_STRINGX4_TO_BUFFER( S1:= CONCAT(sHead, '_TDEF_4_5' ), S2:='$t', S3:= REAL_TO_STRING( stTABLE.aTDef[4,5] ), S4:='$n', wSize := wSize, pBuffer := pBuffer, wPos := wPos );
F_ADD_STRINGX4_TO_BUFFER( S1:= CONCAT(sHead, '_TDEF_4_6' ), S2:='$t', S3:= REAL_TO_STRING( stTABLE.aTDef[4,6] ), S4:='$n', wSize := wSize, pBuffer := pBuffer, wPos := wPos );
END_FUNCTION

(* POU FUN/F_CALC_ENGINE_COEF, ST *)
FUNCTION F_CALC_ENGINE_COEF : BOOL
VAR_INPUT
	Cycle : REAL;
END_VAR
VAR_IN_OUT
	Cfg : ST_ENGINE_CFG;
END_VAR
VAR
END_VAR
Cfg.CycleMaxInc_RPM := Cfg.MaxInc_RPM * Cycle;
Cfg.CycleMaxDec_RPM := Cfg.MaxDec_RPM * Cycle;

IF Cfg.Max_RPM <> 0.0 THEN
	Cfg.Boost_K := Cfg.Boost_RPM / Cfg.Max_RPM;
END_IF

IF Cfg.Max_Torque > Cfg.Min_Torque THEN
	Cfg.Inc_RMP_Perc_WOP_K := Cfg.Inc_RMP_Perc_WOP / (100.0*(Cfg.Max_Torque - Cfg.Min_Torque));
	Cfg.Dec_Flow_Perc_WP_K := Cfg.Dec_Flow_Perc_WP / (100.0*(Cfg.Max_Torque - Cfg.Min_Torque));
END_IF
END_FUNCTION

(* POU FUN/F_CALC_PROPULSION_COEF, ST *)
FUNCTION F_CALC_PROPULSION_COEF : BOOL
VAR_IN_OUT
	Cfg : ST_PROPULSION_CFG;
END_VAR
VAR
	i : INT;
	d : REAL;

END_VAR
d := (Cfg.aThrt_V[4] - Cfg.aThrt_V[0]) / 4.0; (*REVERSE*)

Cfg.aThrt_V[1] := Cfg.aThrt_V[0] + d;
Cfg.aThrt_V[2] := Cfg.aThrt_V[1] + d;
Cfg.aThrt_V[3] := Cfg.aThrt_V[2] + d;

d := (Cfg.aThrt_V[10] - Cfg.aThrt_V[6]) / 4.0; (*FORWARD*)

Cfg.aThrt_V[7] := Cfg.aThrt_V[6] + d;
Cfg.aThrt_V[8] := Cfg.aThrt_V[7] + d;
Cfg.aThrt_V[9] := Cfg.aThrt_V[8] + d;

FOR i := 0 TO 9 BY 1 DO

	IF Cfg.aThrt_V[i+1] <> Cfg.aThrt_V[i] THEN

		Cfg.aEng_K[i] := (Cfg.aEng_RPM[i+1] - Cfg.aEng_RPM[i]) / (Cfg.aThrt_V[i+1] - Cfg.aThrt_V[i]);
		Cfg.aEVP_K[i] := (Cfg.aEVP_mA [i+1] - Cfg.aEVP_mA [i]) / (Cfg.aThrt_V[i+1] - Cfg.aThrt_V[i]);

		Cfg.aEng_Off[i] := Cfg.aEng_RPM[i] - Cfg.aThrt_V[i] * Cfg.aEng_K[i];
		Cfg.aEVP_Off[i] := Cfg.aEVP_mA [i] - Cfg.aThrt_V[i] * Cfg.aEVP_K[i];

	ELSE

		Cfg.aEng_K[i] := 0.0;
		Cfg.aEVP_K[i] := 0.0;

		Cfg.aEng_Off[i] := 0.0;
		Cfg.aEVP_Off[i] := 0.0;

	END_IF

END_FOR
END_FUNCTION

(* POU FUN/F_CALC_KEEL_COEF, ST *)
FUNCTION F_CALC_KEEL_COEF : BOOL
VAR_INPUT
END_VAR
VAR_IN_OUT
	Cfg : ST_KEEL_CFG;
END_VAR
VAR
END_VAR
IF CFG.EVP_Out_Eng_Max <> CFG.EVP_Out_Eng_Min THEN
	CFG.EVP_Out_Fill_K   := (CFG.EVP_Out_Fill_Max - CFG.EVP_Out_Fill_Min) / (CFG.EVP_Out_Eng_Max - CFG.EVP_Out_Eng_Min);
    CFG.EVP_Out_Fill_Off := CFG.EVP_Out_Fill_Min - CFG.EVP_Out_Eng_Min * CFG.EVP_Out_Fill_K;

ELSE
	CFG.EVP_Out_Fill_K   := 0;
    CFG.EVP_Out_Fill_Off := 0;
END_IF
END_FUNCTION

(* POU ALARMS, ST *)
PROGRAM ALARMS
VAR CONSTANT
	UDP_BUF_SIZE  : WORD := 4096;
	TRIG_BUF_SIZE : WORD := 100;
	ALARMS_LIST_SIZE : WORD := 66;
	ALARMS_ARRAY_SIZE : WORD := 203;



END_VAR
VAR
	TankAdver : BOOL;
	EngAdver  : BOOL;
	PumpAdver : BOOL;
	CanAdver: BOOL;

	Clear  : BOOL;
	Buzzer : BOOL;
	Adver  : BOOL;

	LoadTrig : R_TRIG;

	BobStay_adv : BOOL;
	Cylinders_adv : BOOL;
	Special_adv   : BOOL;



	AlarmList : ARRAY[1..ALARMS_LIST_SIZE] OF STRING;
	AlarmFlag : ARRAY[1..ALARMS_LIST_SIZE] OF BOOL;

	AlarmArray : ARRAY[1..ALARMS_ARRAY_SIZE] OF POINTER TO ST_ALARM;

	i : WORD;
	j : WORD;
	SF100x_Mute : BOOL;

	fbUdpSend : FB_UDP_SEND_TRIG;

	aBuffer : ARRAY[0..UDP_BUF_SIZE] OF BYTE;
	wBufPos : DWORD;

	InitArray : BOOL := TRUE;

END_VAR
IF InitArray THEN
	InitArray := FALSE;

	(*Emergency*)
	AlarmArray[ 1] := ADR(SF000.Alarm);

	(*Tank*)
	AlarmArray[ 2] := ADR(SF001.Alarm);
	AlarmArray[ 3] := ADR(SF002.Alarm);
	AlarmArray[ 4] := ADR(SF003.Alarm);
	AlarmArray[ 5] := ADR(SF004.Alarm);
	AlarmArray[ 6] := ADR(SF005.Alarm);
	AlarmArray[ 7] := ADR(SF006.Alarm);
	AlarmArray[ 8] := ADR(SF007.Alarm);
	AlarmArray[ 9] := ADR(SF008.Alarm);
	AlarmArray[10] := ADR(SF009.Alarm);
	AlarmArray[11] := ADR( P010.Alarm);
	AlarmArray[12] := ADR( S011.Alarm);

	(*Pump*)
	AlarmArray[13] := ADR( P001.Alarm);
	AlarmArray[14] := ADR( P002.Alarm);
	AlarmArray[15] := ADR( P051.Alarm);
	AlarmArray[16] := ADR( P052.Alarm);
	AlarmArray[17] := ADR( P101.Alarm);
	AlarmArray[18] := ADR( P103.Alarm);
	AlarmArray[19] := ADR( S101.Alarm);
	AlarmArray[20] := ADR( S102.Alarm);

	(*Engine*)
	AlarmArray[21] := ADR(ENGINE.Alarm1);
	AlarmArray[22] := ADR(ENGINE.Alarm2);
	AlarmArray[23] := ADR(INPUTS.THR_Alarm);
	AlarmArray[24] := ADR(MAIN.fbDE601.Alarm);

	(*Sensors Alarms*)
	AlarmArray[25] := ADR(LS021.Alarm);
	AlarmArray[26] := ADR(LS022.Alarm);
	AlarmArray[27] := ADR(LS023.Alarm);
	AlarmArray[28] := ADR(LS024.Alarm);

	AlarmArray[29] := ADR( P201.Alarm);

	AlarmArray[30] := ADR( P301.Alarm);
	AlarmArray[31] := ADR( P303.Alarm);
	AlarmArray[32] := ADR( P305.Alarm);
	AlarmArray[33] := ADR( P307.Alarm);
	AlarmArray[34] := ADR( P309.Alarm);
	AlarmArray[35] := ADR( P311.Alarm);
	AlarmArray[36] := ADR(LS301.Alarm);
	AlarmArray[37] := ADR(LS303.Alarm);
	AlarmArray[38] := ADR(LS305.Alarm);
	AlarmArray[39] := ADR(LS307.Alarm);
	AlarmArray[40] := ADR(LS309.Alarm);
	AlarmArray[41] := ADR(LS311.Alarm);

	AlarmArray[42] := ADR( P501.Alarm);
	AlarmArray[43] := ADR( P503.Alarm);
	AlarmArray[44] := ADR( P505.Alarm);
	AlarmArray[45] := ADR( P507.Alarm);

	AlarmArray[46] := ADR( P601.Alarm);
	AlarmArray[47] := ADR( P603.Alarm);
	AlarmArray[48] := ADR( P605.Alarm);
	AlarmArray[49] := ADR( P607.Alarm);
	AlarmArray[50] := ADR(LS601.Alarm);
	AlarmArray[51] := ADR(LS605.Alarm);

	AlarmArray[52] := ADR( P701.Alarm);
	AlarmArray[53] := ADR( P703.Alarm);
	AlarmArray[54] := ADR( P705.Alarm);
	AlarmArray[55] := ADR( P707.Alarm);
	AlarmArray[56] := ADR( P709.Alarm);
	AlarmArray[57] := ADR(LS707.Alarm);
	AlarmArray[58] := ADR(LS709.Alarm);

	AlarmArray[59] := ADR(SF801.Alarm);
	AlarmArray[60] := ADR(SF803.Alarm);
	AlarmArray[61] := ADR( P802.Alarm);
	AlarmArray[62] := ADR( P804.Alarm);
	AlarmArray[63] := ADR(LS801.Alarm);
	AlarmArray[64] := ADR(LS803.Alarm);

(*	AlarmArray[65] := ADR( P901.Alarm);*)
(*	AlarmArray[66] := ADR( P903.Alarm);*)
(*	AlarmArray[67] := ADR(LS901.Alarm);*)
(*	AlarmArray[68] := ADR(LS903.Alarm);*)

	AlarmArray[69] := ADR( P1001.Alarm);
	AlarmArray[70] := ADR( P1002.Alarm);
	AlarmArray[71] := ADR(LS1001.Alarm);
	AlarmArray[72] := ADR(LS1002.Alarm);
	AlarmArray[73] := ADR(SF1002.Alarm);
	AlarmArray[74] := ADR(SF1003.Alarm);
	AlarmArray[75] := ADR(SF1004.Alarm);

	AlarmArray[76] := ADR( P1101.Alarm);
	AlarmArray[77] := ADR( P1102.Alarm);

	AlarmArray[78] := ADR( P1202.Alarm);
	AlarmArray[79] := ADR( P1203.Alarm);
	AlarmArray[80] := ADR( P1204.Alarm);
	AlarmArray[81] := ADR( P1205.Alarm);
	AlarmArray[82] := ADR( P1206.Alarm);
	AlarmArray[83] := ADR( P1207.Alarm);
	AlarmArray[84] := ADR( P1208.Alarm);
	AlarmArray[85] := ADR( P1209.Alarm);
	AlarmArray[86] := ADR( P1210.Alarm);
	AlarmArray[87] := ADR( P1211.Alarm);
	AlarmArray[88] := ADR( P1212.Alarm);
	AlarmArray[89] := ADR( P1213.Alarm);
	AlarmArray[90] := ADR( P1214.Alarm);
	AlarmArray[91] := ADR( P1215.Alarm);
	AlarmArray[92] := ADR( P1216.Alarm);
	AlarmArray[93] := ADR( P1219.Alarm);

	AlarmArray[94] := ADR( P1301.Alarm);
	AlarmArray[95] := ADR( P1302.Alarm);
	AlarmArray[96] := ADR(LS1303.Alarm);

	AlarmArray[ 97] := ADR( P1602.Alarm);
	AlarmArray[ 98] := ADR( P1603.Alarm);
	AlarmArray[ 99] := ADR( P1604.Alarm);
	AlarmArray[100] := ADR( P1605.Alarm);

	AlarmArray[101] := ADR(LS1905.Alarm);

	AlarmArray[102] := ADR(LS2001.Alarm);
	AlarmArray[103] := ADR(LS2005.Alarm);

	AlarmArray[104] := ADR(LS2201.Alarm);

	AlarmArray[105] := ADR(LS2301.Alarm);
	AlarmArray[106] := ADR(LS2305.Alarm);

	AlarmArray[107] := ADR(LS2401.Alarm);
	AlarmArray[108] := ADR(LS2409.Alarm);

	AlarmArray[109] := ADR( P2500.Alarm);
	AlarmArray[110] := ADR(LS2501.Alarm);
	AlarmArray[111] := ADR(LS2505.Alarm);

	(*CAN*)
	AlarmArray[112] := ADR(CAN1.Alarm);
	AlarmArray[113] := ADR(CAN2.Alarm);
	AlarmArray[114] := ADR(CAN3.Alarm);
	AlarmArray[115] := ADR(CAN4.Alarm);
	AlarmArray[116] := ADR(CAN5.Alarm);
	AlarmArray[117] := ADR(NJ1939.Alarm);

	AlarmArray[118] := ADR(N20.Alarm);
	AlarmArray[119] := ADR(N21.Alarm);
	AlarmArray[120] := ADR(N22.Alarm);
	AlarmArray[121] := ADR(N23.Alarm);
	AlarmArray[122] := ADR(N24.Alarm);
	AlarmArray[123] := ADR(N25.Alarm);
	AlarmArray[124] := ADR(N26.Alarm);
	AlarmArray[125] := ADR(N27.Alarm);
	AlarmArray[126] := ADR(N28.Alarm);
	AlarmArray[127] := ADR(N29.Alarm);
	AlarmArray[128] := ADR(N30.Alarm);
	AlarmArray[129] := ADR(N31.Alarm);
	AlarmArray[130] := ADR(N32.Alarm);
	AlarmArray[131] := ADR(N33.Alarm);
	AlarmArray[132] := ADR(N34.Alarm);
	AlarmArray[133] := ADR(N35.Alarm);
	AlarmArray[134] := ADR(N36.Alarm);
	AlarmArray[135] := ADR(N37.Alarm);
	AlarmArray[136] := ADR(N38.Alarm);
	AlarmArray[137] := ADR(N39.Alarm);
	AlarmArray[138] := ADR(N40.Alarm);
	AlarmArray[139] := ADR(N41.Alarm);
	AlarmArray[140] := ADR(N42.Alarm);
	AlarmArray[141] := ADR(N43.Alarm);
	AlarmArray[142] := ADR(N44.Alarm);
	AlarmArray[143] := ADR(N47.Alarm);

	AlarmArray[144] := ADR(N50.Alarm);
	AlarmArray[145] := ADR(N51.Alarm);
	AlarmArray[146] := ADR(N52.Alarm);
	AlarmArray[147] := ADR(N53.Alarm);
	AlarmArray[148] := ADR(N54.Alarm);
	AlarmArray[149] := ADR(N55.Alarm);
	AlarmArray[150] := ADR(N56.Alarm);
	AlarmArray[151] := ADR(N57.Alarm);
	AlarmArray[152] := ADR(N58.Alarm);
	AlarmArray[153] := ADR(N59.Alarm);
	AlarmArray[154] := ADR(N60.Alarm);
	AlarmArray[155] := ADR(N61.Alarm);
	AlarmArray[156] := ADR(N64.Alarm);
	AlarmArray[157] := ADR(N70.Alarm);
	AlarmArray[158] := ADR(N71.Alarm);
	AlarmArray[159] := ADR(N72.Alarm);
	AlarmArray[160] := ADR(N73.Alarm);
	AlarmArray[161] := ADR(N74.Alarm);

	AlarmArray[162] := ADR(N102.Alarm);
	AlarmArray[163] := ADR(N103.Alarm);
	AlarmArray[164] := ADR(N104.Alarm);
	AlarmArray[165] := ADR(N105.Alarm);
	AlarmArray[166] := ADR(N106.Alarm);
	AlarmArray[167] := ADR(N107.Alarm);
	AlarmArray[168] := ADR(N108.Alarm);
	AlarmArray[169] := ADR(N109.Alarm);
	AlarmArray[170] := ADR(N110.Alarm);
	AlarmArray[171] := ADR(N111.Alarm);
	AlarmArray[172] := ADR(N112.Alarm);
	AlarmArray[173] := ADR(N113.Alarm);
	AlarmArray[174] := ADR(N114.Alarm);
	AlarmArray[175] := ADR(N115.Alarm);
	AlarmArray[176] := ADR(N116.Alarm);
	AlarmArray[177] := ADR(N117.Alarm);
	AlarmArray[178] := ADR(N118.Alarm);
	AlarmArray[179] := ADR(N119.Alarm);

	AlarmArray[188] := ADR(N10.Alarm);
	AlarmArray[189] := ADR(N11.Alarm);
	AlarmArray[190] := ADR(N12.Alarm);
	AlarmArray[191] := ADR(N13.Alarm);
	AlarmArray[198] := ADR(N20_2.Alarm);

	AlarmArray[200] := ADR(MAIN.fbTackValve.Alarm);

	(*AlarmArray[201] := ADR(SF100.Alarm);*)
	AlarmArray[202] := ADR(S1100.Alarm);

END_IF

LoadTrig(CLK:= PARAMS.Loaded);

IF NOT PARAMS.Loaded OR LoadTrig.Q THEN
	Clear := TRUE;

END_IF

TankAdver := SF001.Alarm.Adver
		  OR SF002.Alarm.Adver
		  OR SF003.Alarm.Adver
		  OR SF004.Alarm.Adver
		  OR SF005.Alarm.Adver
		  OR SF006.Alarm.Adver
		  OR SF007.Alarm.Adver
		  OR SF008.Alarm.Adver
		  OR SF009.Alarm.Adver
		  OR  P010.Alarm.Adver
		  OR  S011.Alarm.Adver
;
PumpAdver :=  P001.Alarm.Adver
		  OR  P002.Alarm.Adver
		  OR  P051.Alarm.Adver
		  OR  P052.Alarm.Adver
		  OR  P101.Alarm.Adver
		  OR  P103.Alarm.Adver
		  OR  S101.Alarm.Adver
		  OR  S102.Alarm.Adver
;
EngAdver  := ENGINE.Alarm1.Adver
		  OR ENGINE.Alarm2.Adver
		  OR INPUTS.THR_Alarm.Adver
		  OR MAIN.fbDE601.Alarm.Adver
;

CanAdver  := FALSE;


(*Fill Allarms array*)
Buzzer := FALSE;
i := 1;

(*ENABLE ALARM*)
(*Tank Enable*)
IF NOT MAIN.aSys_Enable[1] THEN AlarmList[i] := 'Tank Disabled.'; 				AlarmFlag[i] := TRUE;	i := i + 1; TankAdver := TRUE; END_IF
(*Pump Enable*)
IF NOT MAIN.aSys_Enable[4] THEN AlarmList[i] := 'Engine HP Pump 1 Disabled.'; 	AlarmFlag[i] := TRUE;	i := i + 1; PumpAdver := TRUE; END_IF
IF NOT MAIN.aSys_Enable[5] THEN AlarmList[i] := 'Engine HP Pump 2 Disabled.';	AlarmFlag[i] := TRUE;	i := i + 1; PumpAdver := TRUE; END_IF
IF NOT MAIN.aSys_Enable[6] THEN AlarmList[i] := 'PowerPack 1 Disabled.'; 		AlarmFlag[i] := TRUE;	i := i + 1; PumpAdver := TRUE; END_IF
IF NOT MAIN.aSys_Enable[7] THEN AlarmList[i] := 'PowerPack 2 Disabled.'; 		AlarmFlag[i] := TRUE;	i := i + 1; PumpAdver := TRUE; END_IF
(*Engine Enable*)
IF NOT MAIN.aSys_Enable[8] THEN AlarmList[i] := 'Engine Disabled.'; 			AlarmFlag[i] := TRUE;	i := i + 1; EngAdver := TRUE; END_IF
IF NOT MAIN.aSys_Enable[9] THEN AlarmList[i] := 'Propulsion Disabled.'; 		AlarmFlag[i] := TRUE; 	i := i + 1; EngAdver := TRUE; END_IF
(*HP Function Enable*)
IF NOT MAIN.aHP_Enable[ 1] THEN AlarmList[i] := 'TackPort Disabled.';			AlarmFlag[i] := TRUE;	i := i + 1; END_IF
IF NOT MAIN.aHP_Enable[ 2] THEN AlarmList[i] := 'TackStbd Disabled.';			AlarmFlag[i] := TRUE;	i := i + 1; END_IF
IF NOT MAIN.aHP_Enable[ 3] THEN AlarmList[i] := 'J5 Disabled.';					AlarmFlag[i] := TRUE;	i := i + 1; END_IF
IF NOT MAIN.aHP_Enable[ 4] THEN AlarmList[i] := 'J4 Disabled.';					AlarmFlag[i] := TRUE;	i := i + 1; END_IF
IF NOT MAIN.aHP_Enable[ 5] THEN AlarmList[i] := 'Forastay Disabled.';			AlarmFlag[i] := TRUE;	i := i + 1; END_IF
IF NOT MAIN.aHP_Enable[ 6] THEN AlarmList[i] := 'J2 Disabled.';					AlarmFlag[i] := TRUE;	i := i + 1; END_IF
IF NOT MAIN.aHP_Enable[ 7] THEN AlarmList[i] := 'JibInOut Disabled.';			AlarmFlag[i] := TRUE;	i := i + 1; END_IF
IF NOT MAIN.aHP_Enable[ 8] THEN AlarmList[i] := 'JibUpDw Disabled.';			AlarmFlag[i] := TRUE;	i := i + 1; END_IF
(*IF NOT MAIN.aHP_Enable[ 9] THEN AlarmList[i] := 'Vang Disabled.';				AlarmFlag[i] := TRUE;	i := i + 1; END_IF*)
IF NOT MAIN.aHP_Enable[10] THEN AlarmList[i] := 'PropUpDW Disabled.';			AlarmFlag[i] := TRUE;	i := i + 1; END_IF
IF NOT MAIN.aHP_Enable[11] THEN AlarmList[i] := 'TrimTab Disabled.';			AlarmFlag[i] := TRUE;	i := i + 1; END_IF
IF NOT MAIN.aHP_Enable[12] THEN AlarmList[i] := 'Runner Disabled.';				AlarmFlag[i] := TRUE;	i := i + 1; END_IF
IF NOT MAIN.aHP_Enable[13] THEN AlarmList[i] := 'Checkstay Disabled.';			AlarmFlag[i] := TRUE;	i := i + 1; END_IF
IF NOT MAIN.aHP_Enable[14] THEN AlarmList[i] := 'Innerstay Disabled.';			AlarmFlag[i] := TRUE;	i := i + 1; END_IF
IF NOT MAIN.aHP_Enable[15] THEN AlarmList[i] := 'Outhaul Disabled.';			AlarmFlag[i] := TRUE;	i := i + 1; END_IF
IF NOT MAIN.aHP_Enable[16] THEN AlarmList[i] := 'MainCunn Disabled.';			AlarmFlag[i] := TRUE;	i := i + 1;	END_IF
(*IF NOT MAIN.aHP_Enable[17] THEN AlarmList[i] := 'BackstayPort Disabled.';		AlarmFlag[i] := TRUE;	i := i + 1; END_IF
IF NOT MAIN.aHP_Enable[18] THEN AlarmList[i] := 'BackstayStbd Disabled.';		AlarmFlag[i] := TRUE;	i := i + 1; END_IF*)
IF NOT MAIN.aHP_Enable[19] THEN AlarmList[i] := 'WaterBallast Disabled.';		AlarmFlag[i] := TRUE;	i := i + 1; END_IF
(*LP Function Enable*)
IF NOT MAIN.aLP_Enable[ 4] THEN AlarmList[i] := 'Stbd Primary Winch 1202 Disabled.';	AlarmFlag[i] := TRUE;	i := i + 1; END_IF
IF NOT MAIN.aLP_Enable[ 5] THEN AlarmList[i] := 'Stbd Pit Winch 1204 Disabled.';		AlarmFlag[i] := TRUE;	i := i + 1; END_IF
IF NOT MAIN.aLP_Enable[ 6] THEN AlarmList[i] := 'Main Winch 1206 Disabled.';			AlarmFlag[i] := TRUE;	i := i + 1; END_IF
IF NOT MAIN.aLP_Enable[ 7] THEN AlarmList[i] := 'Port Runner Winch 1208 Disabled.';		AlarmFlag[i] := TRUE;	i := i + 1; END_IF
IF NOT MAIN.aLP_Enable[ 8] THEN AlarmList[i] := 'Port Primary Winch 1210 Disabled.';	AlarmFlag[i] := TRUE;	i := i + 1; END_IF
IF NOT MAIN.aLP_Enable[ 9] THEN AlarmList[i] := 'Port Secondary Winch 1212 Disabled.';	AlarmFlag[i] := TRUE;	i := i + 1; END_IF
IF NOT MAIN.aLP_Enable[10] THEN AlarmList[i] := 'Port Pit Winch 1214 Disabled.';		AlarmFlag[i] := TRUE;	i := i + 1; END_IF
IF NOT MAIN.aLP_Enable[11] THEN AlarmList[i] := 'DGBD Disabled.';						AlarmFlag[i] := TRUE;	i := i + 1; END_IF

IF NOT MAIN.aLP_Enable[13] THEN AlarmList[i] := 'Keel Disabled.';						AlarmFlag[i] := TRUE;	i := i + 1; END_IF
IF NOT MAIN.aLP_Enable[14] THEN AlarmList[i] := 'Stbd Runner Winch 1602 Disabled.';		AlarmFlag[i] := TRUE;	i := i + 1; END_IF
IF NOT MAIN.aLP_Enable[15] THEN AlarmList[i] := 'Stbd Secondary Winch 1604 Disabled.';	AlarmFlag[i] := TRUE;	i := i + 1; END_IF
IF NOT MAIN.aLP_Enable[16] THEN AlarmList[i] := 'Traveller Disabled.';					AlarmFlag[i] := TRUE;	i := i + 1; END_IF
IF NOT MAIN.aLP_Enable[17] THEN AlarmList[i] := 'BowThruster Disabled.';				AlarmFlag[i] := TRUE;	i := i + 1; END_IF
IF NOT MAIN.aLP_Enable[18] THEN AlarmList[i] := 'BowThrusterUpDw Disabled.';			AlarmFlag[i] := TRUE;	i := i + 1; END_IF

(*ENGINE Forced Values*)
IF ENGINE.Alarm3 <> ''		THEN AlarmList[i] := ENGINE.Alarm3;        			AlarmFlag[i] := TRUE; 	i := i + 1; EngAdver := TRUE; END_IF

(*WATER BALLAST*)
IF MAIN.fbWB.Error > 0 		THEN AlarmList[i] := CONCAT('Water Ballast Error: ', WORD_TO_STRING(MAIN.fbWB.Error)); AlarmFlag[i] := FALSE; i := i + 1; END_IF

(*COPY TO VISU LIST*)
FOR j := 1 TO ALARMS_ARRAY_SIZE BY 1 DO

	IF AlarmArray[j] <> 0 THEN

		IF AlarmArray[j]^.Adver AND i < ALARMS_LIST_SIZE THEN
			AlarmList[i] := CONCAT( AlarmArray[j]^.TimeInit, ' - ');
			AlarmList[i] := CONCAT( AlarmList[i], AlarmArray[j]^.Text);

			IF AlarmArray[j]^.Alarm THEN
				AlarmList[i] := CONCAT( AlarmList[i], ' - ' );
				AlarmList[i] := CONCAT( AlarmList[i], REAL_TO_STRING(REAL_TO_INT(AlarmArray[j]^.AlLen * 10.0) / 10.0) );
				AlarmList[i] := CONCAT( AlarmList[i], 's' );

			ELSE
				AlarmList[i] := CONCAT( AlarmList[i], ' - ' );
				AlarmList[i] := CONCAT( AlarmList[i], WORD_TO_STRING(AlarmArray[j]^.AlCnt) );
				AlarmList[i] := CONCAT( AlarmList[i], ' times' );

			END_IF

			AlarmFlag[i] := AlarmArray[j]^.Alarm;
			i := i + 1;

		END_IF
	END_IF
END_FOR

(*BUZZER*)
SF100x_Mute := SF100x_Mute AND (SF1003.Alarm.Alarm OR SF1004.Alarm.Alarm);

Buzzer := Buzzer
	OR MAIN.fbDE601.Alarm.Alarm
	OR NOT SF100x_Mute AND (SF1003.Alarm.Alarm OR SF1004.Alarm.Alarm);

Adver  := i > 1;(* OR fbUdpSend.bError;*)

(*Clear unused alarm string*)
FOR i := i TO ALARMS_LIST_SIZE BY 1 DO
	AlarmList[i] := '';
	AlarmFlag[i] := FALSE;
END_FOR

Buzzer := PARAMS.Loaded AND( Buzzer OR TANK.Buzzer OR POWERPACK.Buzzer OR ENGINE.Buzzer );

(*UDP STREAMING*)
IF TOFARO.bCloseAll THEN
	fbUdpSend( bEnable:= FALSE );
END_IF

(*Reset Flag*)
fbUdpSend(
	bEnable:= TRUE,
	bFlag  := FALSE
);

IF fbUDPSend.eStep = UDP_STATE_IDLE AND fbUDPSend.bCreated THEN
	wBufPos := 0;

	FOR j := 1 TO ALARMS_ARRAY_SIZE BY 1 DO

		IF AlarmArray[j] <> 0 THEN

			IF AlarmArray[j]^.AlInit THEN
				AlarmArray[j]^.AlInit := FALSE;

				F_ADD_STRINGX2_TO_BUFFER( S1:= AlarmArray[j]^.TimeInit, S2:= '$t1$t'  , wSize := UDP_BUF_SIZE, pBuffer := ADR(aBuffer), wPos := wBufPos );
				F_ADD_STRINGX2_TO_BUFFER( S1:= AlarmArray[j]^.Text,     S2:= '$t0$r$n', wSize := UDP_BUF_SIZE, pBuffer := ADR(aBuffer), wPos := wBufPos );

				fbUdpSend.bFlag := TRUE;
			END_IF

			IF AlarmArray[j]^.AlEnd THEN
				AlarmArray[j]^.AlEnd := FALSE;

				F_ADD_STRINGX2_TO_BUFFER( S1:= AlarmArray[j]^.TimeEnd, 				 S2:= '$t0$t', wSize := UDP_BUF_SIZE, pBuffer := ADR(aBuffer), wPos := wBufPos );
				F_ADD_STRINGX2_TO_BUFFER( S1:= AlarmArray[j]^.Text,    				 S2:= '$t'   , wSize := UDP_BUF_SIZE, pBuffer := ADR(aBuffer), wPos := wBufPos );
				F_ADD_STRINGX2_TO_BUFFER( S1:= REAL_TO_STRING(AlarmArray[j]^.AlLen), S2:= '$r$n' , wSize := UDP_BUF_SIZE, pBuffer := ADR(aBuffer), wPos := wBufPos );

				fbUdpSend.bFlag := TRUE;
			END_IF

		END_IF
	END_FOR

	fbUdpSend(
		bEnable    := TRUE,
		sRemoteHost:= PARAMS.sUDPAlarmsHost,
		nRemotePort:= PARAMS.nUDPAlarmsPort,
		pBuffer    := ADR(aBuffer),
		wBufLen    := wBufPos,
	);
END_IF
END_PROGRAM

(* POU ENGINE, ST *)
PROGRAM ENGINE
VAR
	fbEngine     : FB_ENGINE;
	fbPropulsion : FB_PROPULSION;

	Propulion_ON : BOOL;
	Pump_ON      : BOOL;
	Engine_ON    : BOOL; (*Con delay*)
	Engine_STOP  : BOOL;
	ForcedRPM    : BOOL;

	ForcedProp     : BOOL;
	ForcedProp_Thr : REAL;
	ForcedProp_Tgt : REAL;
	ForcedProp_Inc : REAL := 0.5; (*0.5V/s - 8 sec full throttle*)

	OldCount : DWORD;
	ErrCount : DWORD;

	SIEngStop  : FB_SMART_INPUT;

	Alarm1 : ST_ALARM;
	Alarm2 : ST_ALARM;
	Alarm3 : STRING;
	Buzzer : BOOL;

	EngineAlCnt : REAL;

	S100_Mute  : BOOL;
	SF100_Mute : BOOL;
	S1100_Mute : BOOL;


END_VAR
IF ALARMS.Clear THEN
	Alarm1.Alarm := FALSE;
	Alarm1.Adver := FALSE;
	Alarm1.AlCnt := 0;
	Alarm1.AlLen := 0.0;

	Alarm2.Alarm := FALSE;
	Alarm2.Adver := FALSE;
	Alarm2.AlCnt := 0;
	Alarm2.AlLen := 0.0;

END_IF

S100_Mute  := S100_Mute   AND  S100.Alarm.Alarm;
SF100_Mute := SF100_Mute  AND  SF100.Alarm.Alarm;
S1100_Mute := S1100_Mute  AND  S1100.AlLow;


(*Alarm Input from engine*)
IF N0_DI4 THEN
	IF NOT Alarm1.Alarm THEN
		Alarm1.AlCnt  := Alarm1.AlCnt + 1;
		Alarm1.AlLen  := 0.0;
		Alarm1.TimeInit := INPUTS.sLocal;
		Alarm1.AlInit   := TRUE;

		Alarm1.Text   := 'Engine Alarm! ';

	ELSE
		Alarm1.AlLen  := Alarm1.AlLen + MAIN.Cycle_Time;

	END_IF

	Alarm1.Adver := TRUE;
	Alarm1.Alarm := TRUE;

	EngineAlCnt  := 0;

ELSIF EngineAlCnt > 5.0 THEN
	IF Alarm1.Alarm THEN
		Alarm1.TimeEnd := INPUTS.sLocal;
		Alarm1.AlEnd   := TRUE;

	END_IF

	Alarm1.Alarm := FALSE;

ELSE
	EngineAlCnt := EngineAlCnt + MAIN.Cycle_Time;

END_IF


SIEngStop(In:= N112_IN.6, T_Cont:= T#500ms, T_DClk:= T#0ms);

(*FLAGS/DIAGNOSIS*)
IF RECV_J1939.F004.Count <> OldCount AND RECV_J1939.F004.EngineActualSpeed > 500.0 THEN
	OldCount := RECV_J1939.F004.Count;
	ErrCount := 0;

	Engine_ON := TRUE;

ELSIF ErrCount > 50 THEN
	Engine_ON := FALSE;

ELSE
	ErrCount := ErrCount + 1;

END_IF

(*STOP*)
IF MAIN.fbTackValve.StopEngine THEN
	Engine_STOP := TRUE;

	IF NOT Alarm2.Alarm THEN
		Alarm2.AlCnt  := Alarm2.AlCnt + 1;
		Alarm2.AlLen  := 0.0;
		Alarm2.TimeInit := INPUTS.sLocal;
		Alarm2.AlInit   := TRUE;

		Alarm2.Text   := 'Engine Stopped by Tack Valves!';

	ELSE
		Alarm2.AlLen  := Alarm2.AlLen + MAIN.Cycle_Time;

	END_IF

	Alarm2.Adver := TRUE;
	Alarm2.Alarm := TRUE;

ELSIF Engine_ON AND RECV_J1939.F004.EngineActualSpeed > PARAMS.stEngineCfg.Stop_RPM THEN
	Engine_STOP := TRUE;

	IF NOT Alarm2.Alarm THEN
		Alarm2.AlCnt  := Alarm2.AlCnt + 1;
		Alarm2.AlLen  := 0.0;
		Alarm2.TimeInit := INPUTS.sLocal;
		Alarm2.AlInit   := TRUE;

		Alarm2.Text   := 'Engine Stopped by Excessive RPM!';

	ELSE
		Alarm2.AlLen  := Alarm2.AlLen + MAIN.Cycle_Time;

	END_IF

	Alarm2.Adver := TRUE;
	Alarm2.Alarm := TRUE;


ELSIF SIEngStop.Event = INIT_CONTINUOUS THEN
	Engine_STOP := TRUE;

	IF NOT Alarm2.Alarm THEN
		Alarm2.AlCnt  := Alarm2.AlCnt + 1;
		Alarm2.AlLen  := 0.0;
		Alarm2.TimeInit := INPUTS.sLocal;
		Alarm2.AlInit   := TRUE;

		Alarm2.Text   := 'Engine Stopped by Stop Button!';

	ELSE
		Alarm2.AlLen  := Alarm2.AlLen + MAIN.Cycle_Time;

	END_IF

	Alarm2.Adver := TRUE;
	Alarm2.Alarm := TRUE;

ELSIF SIEngStop.Event = END_CONTINUOUS THEN
	Engine_STOP := FALSE;

	IF Alarm2.Alarm THEN
		Alarm2.TimeEnd := INPUTS.sLocal;
		Alarm2.AlEnd   := TRUE;

	END_IF

	Alarm2.Alarm := FALSE;

END_IF

Propulion_ON := Engine_ON AND NOT ENGINE.fbPropulsion.Idle;
Pump_ON := PARAMS.Loaded AND NOT( Propulion_ON AND TANK.Reduced );

Alarm3 := '';

IF ForcedProp AND PARAMS.stEngineCfg.EnForceTHR THEN

	Alarm3 := 'Forced Engine THROTTLE! ';

	IF ForcedProp_Thr > 0 THEN
		ForcedProp_Tgt := ForcedProp_Tgt + ForcedProp_Inc * MAIN.Cycle_Time;
		ForcedProp_Tgt := MIN(ForcedProp_Tgt, ForcedProp_Thr);
		ForcedProp_Tgt := MAX(ForcedProp_Tgt, 0.0);

	ELSIF ForcedProp_Thr < 0 THEN
		ForcedProp_Tgt := ForcedProp_Tgt - ForcedProp_Inc * MAIN.Cycle_Time;
		ForcedProp_Tgt := MAX(ForcedProp_Tgt, ForcedProp_Thr);
		ForcedProp_Tgt := MIN(ForcedProp_Tgt, 0.0);

	ELSE
		ForcedProp_Tgt := 0.0;

	END_IF

	THR_Prop     := ForcedProp_Tgt;
	THR_Prop_Err := FALSE;

ELSE
	ForcedProp     := FALSE;
	ForcedProp_Thr := THR_Prop;
	ForcedProp_Tgt := 0.0;

END_IF

(*PROPULSION*)
fbPropulsion(
	Enable    := MAIN.aSys_Enable[9] AND TANK.Enable AND MAIN.aSys_Enable[3],
	Ready     := Engine_ON AND MAIN.fbDE601.PROP_DW,

	Throttle_V   := THR_Prop,
	Throttle_err := THR_Prop_Err,

	Cfg  := PARAMS.stPropulsionCfg,

	FwdEVP => EVP002,
	RevEVP => EVP001,
	MoveEV => EV1101,
);

IF NOT EV1101 THEN
	EVP001 := MAIN.fbKeel.EVP_Eng_I;  (*Verificar estos 2*)
	EVP002 := MAIN.fbKeel.EVP_Eng_O;  (*Verificar estos 2*)
END_IF

(*ENGINE*)
fbEngine(
	Enable := MAIN.aSys_Enable[8] AND TANK.Enable,
	Boost  := FALSE,
	Forced := ForcedRPM AND PARAMS.stEngineCfg.EnForceRPM,

	Hydraulic_RPM  := POWERPACK.TgtRPM,
	Propulsion_RPM := fbPropulsion.Tgt_RPM,
	ActualTorque   := RECV_J1939.F004.EngineActualTorque,

	Cfg            := PARAMS.stEngineCfg,
);

IF ForcedRPM AND PARAMS.stEngineCfg.EnForceRPM THEN
	Alarm3 := CONCAT(Alarm3, 'Forced Engine RPM! ');
ELSE
	ForcedRPM := FALSE;
END_IF

Buzzer := Alarm1.Alarm
	   (*OR NOT SF100_Mute AND SF100.Alarm.Alarm*)
	   OR NOT S1100_Mute AND S1100.AlHig
	   OR S1100.AlMax;
END_PROGRAM

(* POU FB/FB_ENGINE, ST *)
FUNCTION_BLOCK FB_ENGINE
VAR_INPUT
	Enable : BOOL;
	Boost  : BOOL;
	Forced : BOOL;

	Hydraulic_RPM  : REAL;
	Propulsion_RPM : REAL;
	Forced_RPM     : REAL;
	ActualTorque   : REAL;
END_VAR
VAR_IN_OUT
	Cfg : ST_ENGINE_CFG;
END_VAR
VAR_OUTPUT
	Engine_RPM : REAL;
	Available_Perc : REAL;
END_VAR
VAR
	Man_RPM : REAL;
	Use_Man : BOOL;
	Tgt_RPM : REAL;
	Dif_RPM : REAL;
	CyclCnt : REAL;

END_VAR
IF Propulsion_RPM > 0 THEN
	(*Boost Logic*)
	IF Boost THEN
		Tgt_RPM := Propulsion_RPM * Cfg.Boost_K;
	ELSE
		Tgt_RPM := Propulsion_RPM;
	END_IF

	IF ActualTorque > Cfg.Min_Torque THEN
		Available_Perc := 1 - Cfg.Dec_Flow_Perc_WP_K * (ActualTorque - Cfg.Min_Torque);
	ELSE
		Available_Perc := 1;
	END_IF

	(*Valvula = 0*)

ELSIF Hydraulic_RPM > 0 THEN

	IF Hydraulic_RPM >= Tgt_RPM THEN
		CyclCnt := 0;
		Tgt_RPM := Hydraulic_RPM;
	ELSIF CyclCnt >= Cfg.DlyDec_sec THEN
		Tgt_RPM := Hydraulic_RPM;
	ELSE
		CyclCnt := CyclCnt + Cfg.Cycle;
	END_IF

	Available_Perc := 1;

	IF ActualTorque > Cfg.Min_Torque THEN
		Tgt_RPM := Hydraulic_RPM + Hydraulic_RPM * Cfg.Inc_RMP_Perc_WOP_K * (ActualTorque - Cfg.Min_Torque);
	END_IF

(*Valvula = 0*)
ELSE
	Available_Perc := 1;

	IF CyclCnt >= Cfg.DlyDec_sec THEN
		Tgt_RPM := 0;
	ELSE
		CyclCnt := CyclCnt + Cfg.Cycle;
	END_IF

	(*si RPM esta en el rango , Valvula = X*)
END_IF

IF Forced AND Propulsion_RPM = 0 THEN
	Tgt_RPM := MAX(Tgt_RPM, Forced_RPM);

	(*Si tampoco Hydraulic_RPM activo la valvula si RPM esta en el rango

	Por defecto desactivado, hacer que hay que activarlo.
*)

END_IF

(*Ramp*)
Dif_RPM := Tgt_RPM - Engine_RPM;

IF Dif_RPM > Cfg.CycleMaxInc_RPM THEN
	Dif_RPM := Cfg.CycleMaxInc_RPM;

ELSIF Dif_RPM < -Cfg.CycleMaxDec_RPM THEN
	Dif_RPM := -Cfg.CycleMaxDec_RPM;

END_IF

(*Limits*)
IF Boost AND Propulsion_RPM > 0
THEN Engine_RPM := MAX(MIN((Engine_RPM + Dif_RPM), Cfg.Boost_RPM), Cfg.Min_RPM);
ELSE Engine_RPM := MAX(MIN((Engine_RPM + Dif_RPM), Cfg.Max_RPM  ), Cfg.Min_RPM);
END_IF
END_FUNCTION_BLOCK

(* POU FB/FB_PROPULSION, ST *)
FUNCTION_BLOCK FB_PROPULSION
VAR_INPUT
	Enable : BOOL;
	Ready  : BOOL;

	Throttle_V   : REAL;
	Throttle_err : BOOL;
END_VAR
VAR_IN_OUT
	Cfg : ST_PROPULSION_CFG;
END_VAR
VAR_OUTPUT
	Tgt_RPM : REAL;
	FwdEVP  : UINT;
	RevEVP  : UINT;
	MoveEV  : BOOL;
	Idle    : BOOL;
END_VAR
VAR
	State   : WORD;
	IntPos  : DWORD;
	TimeCnt : REAL;
END_VAR
IF NOT Enable THEN
	Tgt_RPM := 0;
	FwdEVP  := 0;
	RevEVP  := 0;
	MoveEV  := FALSE;
	Idle    := TRUE;
	TimeCnt := 0;
	State   := 0;
	RETURN;
END_IF

(*Working States*)
CASE State OF

0: (*Init State: Safety that init with throttle in zero*)
	Tgt_RPM := 0.0;
	FwdEVP  := 0;
	RevEVP  := 0;
	MoveEV  := FALSE;
	Idle    := TRUE;
	TimeCnt := 0;
	
	IF ABS(Throttle_V - Cfg.aThrt_V[5]) < Cfg.IdleDB_V AND NOT Throttle_err THEN
		State := 10;
	END_IF

10: (*Normal Working Mode*)
	IF ABS(Throttle_V - Cfg.aThrt_V[5]) < Cfg.IdleDB_V OR Throttle_err OR NOT Ready THEN
		Tgt_RPM := 0.0;
		FwdEVP  := 0;
		RevEVP  := 0;
	
		IF TimeCnt > CFG.Delay_Off THEN
			MoveEV  := FALSE;
		ELSE
			MoveEV  := TRUE;
			TimeCnt := TimeCnt + CFG.Cycle;
		END_IF
	
		Idle    := TRUE;
	
	ELSE
		IF Throttle_V <= Cfg.aThrt_V[0] THEN (*REVERSE*)
	  		Tgt_RPM := cfg.aEng_RPM[0];
			FwdEVP  := 0;
			RevEVP  := REAL_TO_UINT(cfg.aEVP_mA [0]);
			MoveEV  := TRUE;
	
		ELSIF Throttle_V >= Cfg.aThrt_V[10] THEN (*FORWARD*)
	    	Tgt_RPM := cfg.aEng_RPM[10];
			FwdEVP  := REAL_TO_UINT(cfg.aEVP_mA [10]);
			RevEVP  := 0;
			MoveEV  := TRUE;
	
		ELSE
	  		IntPos := F_LOCATE_IN_BUFFER( Value:= Throttle_V, Buffer:= ADR(Cfg.aThrt_V[0]), Size:= 11 );
	
			IF Throttle_V < Cfg.aThrt_V[5] THEN (*REVERSE*)
				Tgt_RPM := Throttle_V * Cfg.aEng_K[IntPos] + Cfg.aEng_Off[IntPos];
				FwdEVP  := 0;
				RevEVP  := REAL_TO_UINT(Throttle_V * Cfg.aEVP_K[IntPos] + Cfg.aEVP_Off[IntPos]);
				MoveEV  := TRUE;
	
			ELSE (*FORWARD*)
				Tgt_RPM := Throttle_V * Cfg.aEng_K[IntPos] + Cfg.aEng_Off[IntPos];
				FwdEVP  := REAL_TO_UINT(Throttle_V * Cfg.aEVP_K[IntPos] + Cfg.aEVP_Off[IntPos]);
				RevEVP  := 0;
				MoveEV  := TRUE;
	
			END_IF
	    END_IF
	
		TimeCnt := 0.0;
		Idle    := FALSE;

	END_IF

END_CASE
END_FUNCTION_BLOCK

(* POU RECV_J1939, ST *)
PROGRAM RECV_J1939
VAR
	i: INT;
	State : WORD;

	F003: FB_DECODE_F003;
	F004: FB_DECODE_F004;
	FEDB: FB_DECODE_FEDB;
	FEE5: FB_DECODE_FEE5;
	FEEE: FB_DECODE_FEEE;
	FEEF: FB_DECODE_FEEF;
	FEF2: FB_DECODE_FEF2;
	FEF6: FB_DECODE_FEF6;
	FEF7: FB_DECODE_FEF7;

	RxFrame: VARTYPE_EXTCANQUEUE;
	MaskID : DWORD;

	rxData: ARRAY [0..7] OF USINT; (*for debug*)


(*VISUALIZATION*)
(*	 vF003 : CobIdDataVisualize;
	strF003 : STRING;
	 vF004 : CobIdDataVisualize;
	strF004 : STRING;
	 vFEEE : CobIdDataVisualize;
	strFEEE : STRING;
*)
END_VAR
(*Receiving block*)
IF J1939_Outputs.RxCounter <> J1939_Inputs.RxCounter THEN
	FOR i := 0 TO (J1939_Inputs.NoOfRxMessages-1) BY 1 DO
		MEMCPY( destAddr := ADR(RxFrame.length ), srcAddr := ADR(J1939_Inputs.RxMessages[i]), n := 14 );

		MaskID := RxFrame.cobId AND 16#01FFFF00;

		(*Case structure to catch specific CobId and parse data from it*)
		CASE MaskID OF

		16#00F00400:(*Electronic Engine Controller 1: EEC1, every 20ms*)
			F004( IN:= RxFrame.RxData );
			(*vF004(rxData:=ADR(RxFrame.RxData) , strRxData=>strF004 );*)

		16#00F00300: (*Electronic Engine Controller 2: EEC2, every 50ms*)
			F003( IN:= RxFrame.RxData );
			(*vF003(rxData:=ADR(RxFrame.RxData) , strRxData=>strF003 );*)

		16#00FEDB00: (*Engine Injector Metering Rail 1 Pressure, every 500ms*)
			FEDB( IN:= RxFrame.RxData );

		16#00FEE500: (*Engine Hours, Revolutions HOURS, *)
			FEE5( IN:= RxFrame.RxData );

		16#00FEEE00: (*Engine Temperature, every 1000ms*)
			FEEE( IN:= RxFrame.RxData );

		16#00FEEF00: (*Engine Fluid Level / Pressure, every 100ms*)
			FEEF( IN:= RxFrame.RxData );

		16#00FEF200: (*Fuel Economy (Liquid) LFE1, every 500ms*)
			FEF2( IN:= RxFrame.RxData );

		16#00FEF600: (*Inlet / Exhaust Conditions #1: IEC1, every 500ms*)
			FEF6( IN:= RxFrame.RxData );

		16#00FEF700: (*Vehicle Electrical Power, every 1000ms*)
			FEF7( IN:= RxFrame.RxData );

			(*MEMCPY( destAddr := ADR(rxData), srcAddr := ADR(RxFrame.RxData), n := 8 );*)


		END_CASE
	END_FOR

	J1939_Outputs.RxCounter := J1939_Outputs.RxCounter+1;
END_IF

State := CAN1_State;
State := State AND 16#00FF;
END_PROGRAM

(* POU PGN FB/FB_DECODE_F003, ST *)
FUNCTION_BLOCK FB_DECODE_F003
VAR_IN_OUT
	IN: ARRAY [0..7] OF USINT;
END_VAR
VAR_OUTPUT
	Satus              : BYTE;
	AccPedalPosition   : REAL;
	LoadAtCurrentSpeed : USINT;

	Count : DWORD;
END_VAR
VAR
	Debug : BOOL;
	Buffer: ARRAY [0..7] OF USINT;
END_VAR
Satus              := IN[0];
AccPedalPosition   := BUFFER_TO_REAL( pBuffer:= ADR(IN[1]), ByteSize := 1, Scale:= 0.4, Offset := 0.0 );
LoadAtCurrentSpeed := IN[2];

Count := Count + 1;

IF Debug THEN MEMCPY(destAddr := ADR(Buffer), srcAddr := ADR(IN), n := 8); END_IF
END_FUNCTION_BLOCK

(* POU PGN FB/FB_DECODE_F004, ST *)
FUNCTION_BLOCK FB_DECODE_F004
VAR_IN_OUT
	IN: ARRAY [0..7] OF USINT;
END_VAR
VAR_OUTPUT
	EngineTorqueMode    : BYTE;
	DriverDemandTorque  : SINT;
	EngineActualTorque  : SINT;
	EngineActualSpeed	: REAL;
	EngineControlSource : BYTE;
	EngineStarterMode   : BYTE;
	EngineDemandTorque  : SINT;

	Count : DWORD;
END_VAR
VAR
	Debug : BOOL;
	Buffer: ARRAY [0..7] OF USINT;
END_VAR
EngineTorqueMode    := IN[0];
DriverDemandTorque  := IN[1]-125;
EngineActualTorque  := IN[2]-125;
EngineActualSpeed   := BUFFER_TO_REAL( pBuffer:= ADR(IN[3]), ByteSize := 2, Scale:= 0.125, Offset := 0.0 );
EngineControlSource := IN[5];
EngineStarterMode   := IN[6];
EngineDemandTorque  := IN[7]-125;

Count := Count + 1;

IF Debug THEN MEMCPY(destAddr := ADR(Buffer), srcAddr := ADR(IN), n := 8); END_IF
END_FUNCTION_BLOCK

(* POU PGN FB/FB_DECODE_FEDB, ST *)
FUNCTION_BLOCK FB_DECODE_FEDB (*SPN 157 Engine Injector Metering Rail 1 Pressure*)
VAR_IN_OUT
	IN: ARRAY [0..7] OF USINT;
END_VAR
VAR_OUTPUT
	EngineInjectorMeteringRail1Pressure : REAL;

	Count : DWORD;
END_VAR
VAR
	Debug : BOOL;
	Buffer: ARRAY [0..7] OF USINT;
END_VAR
EngineInjectorMeteringRail1Pressure  := BUFFER_TO_REAL( pBuffer:= ADR(IN[2]), ByteSize := 2, Scale:= 0.00390625, Offset:= 0.0 );

Count := Count + 1;

IF Debug THEN MEMCPY(destAddr := ADR(Buffer), srcAddr := ADR(IN), n := 8); END_IF
END_FUNCTION_BLOCK

(* POU PGN FB/FB_DECODE_FEE5, ST *)
FUNCTION_BLOCK FB_DECODE_FEE5
VAR_IN_OUT
	IN: ARRAY [0..7] OF USINT;
END_VAR
VAR_OUTPUT
	EngineTotalHoursOfOperation : REAL;

	Count : DWORD;
END_VAR
VAR
	Debug : BOOL;
	Buffer: ARRAY [0..7] OF USINT;
END_VAR
EngineTotalHoursOfOperation := BUFFER_TO_REAL( pBuffer:= ADR(IN[0]), ByteSize := 4, Scale:= 0.05, Offset:= 0.0 );

Count := Count + 1;

IF Debug THEN MEMCPY(destAddr := ADR(Buffer), srcAddr := ADR(IN), n := 8); END_IF
END_FUNCTION_BLOCK

(* POU PGN FB/FB_DECODE_FEEE, ST *)
FUNCTION_BLOCK FB_DECODE_FEEE
VAR_IN_OUT
	IN: ARRAY [0..7] OF USINT;
END_VAR
VAR_OUTPUT
	EngineCoolantTemperature : REAL;
	EngineFuelTemperature    : REAL;
	EngineOilTemperature     : REAL;
	EngineIntercoolerTemperature : REAL;

	Count : DWORD;
END_VAR
VAR
	Debug : BOOL;
	Buffer: ARRAY [0..7] OF USINT;
END_VAR
EngineCoolantTemperature := IN[0] - 40.0;
EngineFuelTemperature    := IN[1] - 40.0;
EngineOilTemperature     := BUFFER_TO_REAL( pBuffer:= ADR(IN[2]), ByteSize := 2, Scale:= 0.03125, Offset:= -273.0 );
EngineIntercoolerTemperature := IN[6] - 40.0;

Count := Count + 1;

IF Debug THEN MEMCPY(destAddr := ADR(Buffer), srcAddr := ADR(IN), n := 8); END_IF
END_FUNCTION_BLOCK

(* POU PGN FB/FB_DECODE_FEEF, ST *)
FUNCTION_BLOCK FB_DECODE_FEEF (*Engine Fluid Level/Pressure 1 EFL/P1*)
VAR_IN_OUT
	IN: ARRAY [0..7] OF USINT;
END_VAR
VAR_OUTPUT
	FuelDeliveryPressure : REAL;
	EngineOilLevel       : REAL;
	EngineOilPressure    : REAL;
	CrankcasePressure    : REAL;
	CoolantPressure      : REAL;
	CoolantLevel         : REAL;

	Count : DWORD;
END_VAR
VAR
	Debug : BOOL;
	Buffer: ARRAY [0..7] OF USINT;
END_VAR
FuelDeliveryPressure := BUFFER_TO_REAL( pBuffer:= ADR(IN[0]), ByteSize := 1, Scale:= 4.0,       Offset := 0.0 );
EngineOilLevel       := BUFFER_TO_REAL( pBuffer:= ADR(IN[2]), ByteSize := 1, Scale:= 0.4,       Offset := 0.0 );
EngineOilPressure    := BUFFER_TO_REAL( pBuffer:= ADR(IN[3]), ByteSize := 1, Scale:= 4.0,       Offset := 0.0 );
CrankcasePressure    := BUFFER_TO_REAL( pBuffer:= ADR(IN[4]), ByteSize := 2, Scale:= 0.0078125, Offset := -250.0 );
CoolantPressure      := BUFFER_TO_REAL( pBuffer:= ADR(IN[6]), ByteSize := 1, Scale:= 2.0,       Offset := 0.0 );
CoolantLevel         := BUFFER_TO_REAL( pBuffer:= ADR(IN[7]), ByteSize := 1, Scale:= 0.4,       Offset := 0.0 );

Count := Count + 1;

IF Debug THEN MEMCPY(destAddr := ADR(Buffer), srcAddr := ADR(IN), n := 8); END_IF
END_FUNCTION_BLOCK

(* POU PGN FB/FB_DECODE_FEF2, ST *)
FUNCTION_BLOCK FB_DECODE_FEF2
VAR_IN_OUT
	IN: ARRAY [0..7] OF USINT;
END_VAR
VAR_OUTPUT
	EngineFuelRate : REAL;

	Count : DWORD;
END_VAR
VAR
	Debug : BOOL;
	Buffer: ARRAY [0..7] OF USINT;
END_VAR
EngineFuelRate := BUFFER_TO_REAL( pBuffer:= ADR(IN[0]), ByteSize := 2, Scale:= 0.05, Offset := 0.0 );

Count := Count + 1;

IF Debug THEN MEMCPY(destAddr := ADR(Buffer), srcAddr := ADR(IN), n := 8); END_IF
END_FUNCTION_BLOCK

(* POU PGN FB/FB_DECODE_FEF6, ST *)
FUNCTION_BLOCK FB_DECODE_FEF6
VAR_IN_OUT
	IN: ARRAY [0..7] OF USINT;
END_VAR
VAR_OUTPUT
	EngineIntakeMF1Pressure    : REAL;
	EngineIntakeMF1Temperature : REAL;

	Count : DWORD;
END_VAR
VAR
	Debug : BOOL;
	Buffer: ARRAY [0..7] OF USINT;
END_VAR
EngineIntakeMF1Pressure    := BUFFER_TO_REAL( pBuffer:= ADR(IN[1]), ByteSize := 1, Scale:= 2.0, Offset :=   0.0 );
EngineIntakeMF1Temperature := BUFFER_TO_REAL( pBuffer:= ADR(IN[2]), ByteSize := 1, Scale:= 1.0, Offset := -40.0 );

Count := Count + 1;

IF Debug THEN MEMCPY(destAddr := ADR(Buffer), srcAddr := ADR(IN), n := 8); END_IF
END_FUNCTION_BLOCK

(* POU PGN FB/FB_DECODE_FEF7, ST *)
FUNCTION_BLOCK FB_DECODE_FEF7
VAR_IN_OUT
	IN: ARRAY [0..7] OF USINT;
END_VAR
VAR_OUTPUT
	ElectricalPotential : REAL;

	Count : DWORD;
END_VAR
VAR
	Debug : BOOL;
	Buffer: ARRAY [0..7] OF USINT;
END_VAR
ElectricalPotential := BUFFER_TO_REAL( pBuffer:= ADR(IN[6]), ByteSize := 2, Scale:= 0.05, Offset := 0.0 );

Count := Count + 1;

IF Debug THEN MEMCPY(destAddr := ADR(Buffer), srcAddr := ADR(IN), n := 8); END_IF
END_FUNCTION_BLOCK

(* POU TANK, ST *)
PROGRAM TANK
VAR
	Enable : BOOL;
	Buzzer : BOOL;

	Reduced: BOOL; (*Fuerza a las funcones  atrabajar de modo reducido de flujo, Limitacion sobre winches  y sobre el motor?*)
				   (*Solo propulsion o solo hidraulica, y ademas, solo 1 PP*)

	SF002_Mute : BOOL;
	 P010_Mute : BOOL;
	 S011_Mute : BOOL;

	BypassLevel : BOOL;

	TankEnable: BOOL;
END_VAR
SF002_Mute := SF002_Mute AND SF002.Alarm.Alarm;
 P010_Mute := P010_Mute  AND (P010.AlMax OR P010.AlMin);
 S011_Mute := S011_Mute  AND  S011.AlLow;

IF NOT MAIN.aSys_Enable[2] AND NOT MAIN.aSys_Enable[3] THEN
	BypassLevel := FALSE;
END_IF

(*Conclusion*)
Enable := PARAMS.Loaded
	AND NOT SF000.Alarm.Alarm							(*Emergency button*)
	AND NOT SF001.Alarm.Alarm							(*Main Return*)
	AND (NOT SF009.Alarm.Alarm OR  BypassLevel)			(*Level*)
	AND NOT (SF003.Alarm.Alarm AND SF004.Alarm.Alarm) 	(*Return1*)
	AND NOT (SF005.Alarm.Alarm AND SF006.Alarm.Alarm) 	(*Return2*)
	AND NOT (SF007.Alarm.Alarm AND SF008.Alarm.Alarm)	(*Suction*)
	AND NOT (SF007.Alarm.Alarm AND (SF004.Alarm.Alarm OR SF006.Alarm.Alarm))
	AND NOT (SF008.Alarm.Alarm AND (SF003.Alarm.Alarm OR SF005.Alarm.Alarm))
	AND NOT S011.AlMax
;

Enable := Enable AND MAIN.aSys_Enable[1];

Reduced := Enable AND
	 ( SF003.Alarm.Alarm
	OR SF004.Alarm.Alarm
	OR SF005.Alarm.Alarm
	OR SF006.Alarm.Alarm
	OR SF007.Alarm.Alarm
	OR SF008.Alarm.Alarm
);

Buzzer := MAIN.aSys_Enable[1] AND (
	   NOT SF002_Mute AND SF002.Alarm.Alarm
	OR NOT  P010_Mute AND (P010.AlMax OR P010.AlMin)
	OR NOT  S011_Mute AND  S011.AlHig
	OR S011.AlMax
);

(*Enable := TRUE; *)
END_PROGRAM

(* POU POWERPACK, ST *)
PROGRAM POWERPACK
VAR
	fbPP1 : FB_POWERPACK;
	fbPP2 : FB_POWERPACK;

	NHP   : UINT;
	NSF   : UINT;
	NLP   : UINT;
	NW    : UINT;

	LP_Perc  : REAL;

	WinchReady : BOOL;

	LP_RPM  : REAL;
	HP_RPM  : REAL;
	TgtRPM  : REAL;

	PP1_HP : BOOL;
	PP1_LP : BOOL;
	PP2_HP : BOOL;
	PP2_LP : BOOL;

	Buzzer: BOOL;
	Mute  : BOOL;
	Bypass: BOOL;
	PP_Adver : BOOL;
	HP_Adver : BOOL;

	EV1502_Time : REAL;
	(*Calib*)
	Calib1 : BOOL;
	Calib2 : BOOL;
	CalThr : REAL;
	CalMax : REAL := 5.0;
	CalInc : REAL := 0.01;

END_VAR
THR_PP1 := 0.0;
THR_PP2 := 0.0;

KEY_PP1 := FALSE;
KEY_PP2 := FALSE;

EV101 := FALSE;
EV102 := FALSE;
EV103 := FALSE;
EV104 := FALSE;

(*Count Small Functions HP*)
NSF := MAIN.fbDE605.OUT_HP

	 + MAIN.fbWB_A.OUT_HP
	 + MAIN.fbWB_B.OUT_HP
	 + MAIN.fbWB_C.OUT_HP
	 + MAIN.fbWB_D.OUT_HP
	 + MAIN.fbWB_E.OUT_HP
	 + MAIN.fbWB_F.OUT_HP
	 + MAIN.fbWB_G.OUT_HP
	 + MAIN.fbWB_H.OUT_HP
	 + MAIN.fbWB_I.OUT_HP
	 + MAIN.fbWB_J.OUT_HP
	 + MAIN.fbWB_K.OUT_HP
	 + MAIN.fbWB_L.OUT_HP
	 + MAIN.fbWB_M.OUT_HP
	 + MAIN.fbWB_N.OUT_HP
	 + MAIN.fbWB_R.OUT_HP
	 + MAIN.fbWB_S.OUT_HP
	 + MAIN.fbWB_PUD.OUT_HP
	 + MAIN.fbWB_PAF.OUT_HP
	 + MAIN.fbWB_SUD.OUT_HP
	 + MAIN.fbWB_SAF.OUT_HP
;

(*Count All HP*)
NHP := NSF
	 + MAIN.fbSE301.OUT_HP
	 + MAIN.fbSE303.OUT_HP
	 + MAIN.fbSE305.OUT_HP
	 + MAIN.fbSE307.OUT_HP
	 + MAIN.fbSE309.OUT_HP
	 + MAIN.fbSE311.OUT_HP
	 + MAIN.fbSE501.OUT_HP
	 + MAIN.fbSE503.OUT_HP
	 + MAIN.fbSE505.OUT_HP
	 + MAIN.fbDE601.OUT_HP
(*	 + MAIN.fbDE605.OUT_HP*)
	 + MAIN.fbSE701.OUT_HP
	 + MAIN.fbSE703.OUT_HP
	 + MAIN.fbSE705.OUT_HP
	 + MAIN.fbSE707.OUT_HP
	 + MAIN.fbSE709.OUT_HP

     + MAIN.fbBSY.OUT_HP
(*	 + MAIN.fbSE901.OUT_HP
	 + MAIN.fbSE903.OUT_HP*)

(*	 + MAIN.fbWB_A.OUT_HP
	 + MAIN.fbWB_B.OUT_HP
	 + MAIN.fbWB_C.OUT_HP
	 + MAIN.fbWB_D.OUT_HP
	 + MAIN.fbWB_E.OUT_HP
	 + MAIN.fbWB_F.OUT_HP
	 + MAIN.fbWB_G.OUT_HP
	 + MAIN.fbWB_H.OUT_HP
	 + MAIN.fbWB_I.OUT_HP
	 + MAIN.fbWB_J.OUT_HP
	 + MAIN.fbWB_K.OUT_HP
	 + MAIN.fbWB_L.OUT_HP
	 + MAIN.fbWB_M.OUT_HP
	 + MAIN.fbWB_N.OUT_HP
	 + MAIN.fbWB_R.OUT_HP
	 + MAIN.fbWB_S.OUT_HP
	 + MAIN.fbWB_PUD.OUT_HP
	 + MAIN.fbWB_PAF.OUT_HP
	 + MAIN.fbWB_SUD.OUT_HP
	 + MAIN.fbWB_SAF.OUT_HP *)

	 + MAIN.fbTraveller.OUT_HP
;

(*Count LP*)
NW := MAIN.fbW1202.OUT_LP
	+ MAIN.fbW1204.OUT_LP
	+ MAIN.fbW1206.OUT_LP
	+ MAIN.fbW1208.OUT_LP
	+ MAIN.fbW1210.OUT_LP
	+ MAIN.fbW1212.OUT_LP
	+ MAIN.fbW1214.OUT_LP
	+ MAIN.fbW1602.OUT_LP
	+ MAIN.fbW1604.OUT_LP
;

NLP := NW
	+ MAIN.fbKeel.OUT_LP
	+ MAIN.fbBoard.OUT_LP
	+ MAIN.fbTraveller.OUT_LP

	+ MAIN.fbWB.OUT_LP

	+ MAIN.fbBowThr.OUT_LP
	+ MAIN.fbBowThrUpDw.OUT_LP
;

TgtRPM  := 0.0;
LP_RPM  := 0.0;
HP_RPM  := 0.0;

PP1_HP := FALSE;
PP1_LP := FALSE;
PP2_HP := FALSE;
PP2_LP := FALSE;


IF ENGINE.Engine_ON THEN
	LP_Perc := ENGINE.fbEngine.Available_Perc;

	(*Evaluate HP*)
	CASE NHP OF
	0:
		EV105 := FALSE;
		EV106 := FALSE;

	1:
		IF    MAIN.aSys_Enable[4] THEN EV105 := TRUE;
		ELSIF MAIN.aSys_Enable[5] THEN EV106 := TRUE;
		END_IF

	ELSE
		EV105 := MAIN.aSys_Enable[4];
		EV106 := MAIN.aSys_Enable[5];

	END_CASE

	(*	Any function only PP?? *)

	IF ENGINE.fbPropulsion.Idle THEN
		WinchReady := NW < PARAMS.stEngineCfg.N_Winch_WOP;

		IF NLP > 0 THEN
			IF MAIN.fbKeel.OUT_LP > 0 THEN
				WinchReady := NW < PARAMS.stEngineCfg.N_Winch_WK;
				LP_RPM := PARAMS.stEngineCfg.LP_CK_RPM;

			ELSIF NLP = 1 THEN LP_RPM := PARAMS.stEngineCfg.LP_1x_RPM;
			ELSIF NLP = 2 THEN LP_RPM := PARAMS.stEngineCfg.LP_2x_RPM;
			ELSIF NLP = 3 THEN LP_RPM := PARAMS.stEngineCfg.LP_3x_RPM;
			ELSE               LP_RPM := PARAMS.stEngineCfg.LP_Nx_RPM;
			END_IF
		END_IF

		IF NHP > 0 THEN
			IF NHP = NSF
			THEN HP_RPM := PARAMS.stEngineCfg.HP_SF_RPM;
			ELSE HP_RPM := PARAMS.stEngineCfg.HP_Nx_RPM;
			END_IF
		END_IF

		TgtRPM := MAX(LP_RPM, HP_RPM);

		IF TgtRPM = 0 THEN

		;

		(*
			Si no TgtRPM pero engine tiene RPM tgt interno sea del delay o del forced con el flag.
			comparo rango de RPM y habilito la Valvula 1611
			Tambien valvula 105 y el Link 107 mas abajo.

			Evaluo tambien la logica del EV1501 y EV1502 o igual solo EV1501 porque no tiene que haber presion.

			MEjor si meto una presion mazima medida en P101.
		*)
		END_IF

	ELSE
		WinchReady := NW < PARAMS.stEngineCfg.N_Winch_WP;

		IF MAIN.fbKeel.OUT_LP > 0 THEN
			PP1_LP := fbPP1.Enable;
			PP2_LP := fbPP2.Enable;
		END_IF

	END_IF

	EV1501 := FALSE;
	EV1502 := FALSE;

(*With PowerPack*)
ELSE
	LP_Perc  := 1;
	WinchReady := TRUE;

	(*Evaluate HP*)
	CASE NHP OF
	0:
		PP1_HP := FALSE;
		PP2_HP := FALSE;

	1:
		IF    fbPP1.Enable THEN PP1_HP := TRUE;
		ELSIF fbPP2.Enable THEN PP2_HP := TRUE;
		END_IF

	ELSE
		PP1_HP := fbPP1.Enable;
		PP2_HP := fbPP2.Enable;

	END_CASE

	(*Evaluate LP*)
	CASE NLP OF
	0:
		PP1_LP := FALSE;
		PP2_LP := FALSE;

	(*1:
		IF    fbPP1.Enable THEN PP1_LP := TRUE;
		ELSIF fbPP2.Enable THEN PP2_LP := TRUE;
		END_IF*)

	ELSE
		PP1_LP := fbPP1.Enable;
		PP2_LP := fbPP2.Enable;

	END_CASE

	EV1501 := PP1_LP OR PP2_LP;

	IF EV1501 = TRUE THEN
		EV1502_Time := 1.0;
		EV1502 := FALSE;

	ELSIF EV1502_Time > 0.0 THEN
		EV1502_Time := EV1502_Time - MAIN.Cycle_Time;
		EV1502 := TRUE;

	ELSE
		EV1502 := FALSE;

	END_IF

END_IF

(*POWERPACKS*)
fbPP1(
	Enable := MAIN.aSys_Enable[6] AND TANK.Enable AND (NOT S101.AlMax OR Bypass),

	IN_HP := PP1_HP,
	IN_LP := PP1_LP,

	LP_P := P101,
	HP_P := P103,
	CFG  := PARAMS.stPowerpackCfg,

	OUT_EV_HP => EV103,
	OUT_EV_LP => EV101,
(*	OUT_EV_LNK=> ,*)
	OUT_KEY   => KEY_PP1,
	OUT_THR   => THR_PP1
);

fbPP2(
	Enable := MAIN.aSys_Enable[7] AND TANK.Enable AND (NOT S102.AlMax OR Bypass),

	IN_HP := PP2_HP,
	IN_LP := PP2_LP,

	LP_P := P101,
	HP_P := P103,
	CFG  := PARAMS.stPowerpackCfg,

